LIN {X -0.050,Y -603.917,Z 1305.029,A 0.000,B 0.000,C 90.000,E1 41.148} C_DIS
LIN {X -0.165,Y -603.300,Z 1305.021,A 0.000,B 0.000,C 90.000,E1 39.850} C_DIS
LIN {X 0.003,Y -602.782,Z 1305.016,A 0.000,B 0.000,C 90.000,E1 38.785} C_DIS
LIN {X 0.042,Y -602.471,Z 1305.013,A 0.000,B 0.000,C 90.000,E1 38.257} C_DIS
LIN {X -0.014,Y -601.272,Z 1305.005,A 0.000,B 0.000,C 90.000,E1 36.950} C_DIS
LIN {X 0.141,Y -599.989,Z 1305.000,A 0.000,B 0.000,C 90.000,E1 35.884} C_DIS
LIN {X 0.275,Y -598.512,Z 1304.994,A 0.000,B 0.000,C 90.000,E1 34.818} C_DIS
LIN {X 0.273,Y -596.215,Z 1304.986,A 0.000,B 0.000,C 90.000,E1 33.499} C_DIS
LIN {X -0.207,Y -594.487,Z 1304.982,A 0.000,B 0.000,C 90.000,E1 32.752} C_DIS
LIN {X 0.007,Y -591.783,Z 1304.976,A 0.000,B 0.000,C 90.000,E1 31.671} C_DIS
LIN {X -0.010,Y -589.415,Z 1304.972,A 0.000,B 0.000,C 90.000,E1 30.875} C_DIS
LIN {X -0.049,Y -586.731,Z 1304.967,A 0.000,B 0.000,C 90.000,E1 30.079} C_DIS
LIN {X -0.115,Y -583.665,Z 1304.963,A 0.000,B 0.000,C 90.000,E1 29.283} C_DIS
LIN {X -0.216,Y -580.058,Z 1304.958,A 0.000,B 0.000,C 90.000,E1 28.487} C_DIS
LIN {X 0.289,Y -577.403,Z 1304.955,A 0.000,B 0.000,C 90.000,E1 27.897} C_DIS
LIN {X -0.238,Y -572.396,Z 1304.950,A 0.000,B 0.000,C 90.000,E1 27.001} C_DIS
LIN {X -0.051,Y -569.282,Z 1304.947,A 0.000,B 0.000,C 90.000,E1 26.437} C_DIS
LIN {X 0.274,Y -564.919,Z 1304.943,A 0.000,B 0.000,C 90.000,E1 25.720} C_DIS
LIN {X -0.101,Y -561.279,Z 1304.940,A 0.000,B 0.000,C 90.000,E1 25.207} C_DIS
LIN {X 0.009,Y -557.381,Z 1304.937,A 0.000,B 0.000,C 90.000,E1 24.643} C_DIS
LIN {X 0.090,Y -553.159,Z 1304.934,A 0.000,B 0.000,C 90.000,E1 24.079} C_DIS
LIN {X -0.098,Y -546.387,Z 1304.929,A 0.000,B 0.000,C 90.000,E1 23.259} C_DIS
LIN {X 0.140,Y -539.069,Z 1304.925,A 0.000,B 0.000,C 90.000,E1 22.386} C_DIS
LIN {X 0.134,Y -531.413,Z 1304.920,A 0.000,B 0.000,C 90.000,E1 21.535} C_DIS
LIN {X 0.190,Y -522.299,Z 1304.914,A 0.000,B 0.000,C 90.000,E1 20.556} C_DIS
LIN {X -0.102,Y -511.906,Z 1304.908,A 0.000,B 0.000,C 90.000,E1 19.504} C_DIS
LIN {X -0.036,Y -501.097,Z 1304.902,A 0.000,B 0.000,C 90.000,E1 18.417} C_DIS
LIN {X 0.246,Y -491.595,Z 1304.897,A 0.000,B 0.000,C 90.000,E1 17.457} C_DIS
LIN {X 0.090,Y -484.623,Z 1304.893,A 0.000,B 0.000,C 90.000,E1 16.804} C_DIS
LIN {X -0.137,Y -474.406,Z 1304.888,A 0.000,B 0.000,C 90.000,E1 15.898} C_DIS
LIN {X -0.208,Y -456.704,Z 1304.879,A 0.000,B 0.000,C 90.000,E1 14.300} C_DIS
LIN {X -0.186,Y -437.759,Z 1304.869,A 0.000,B 0.000,C 90.000,E1 12.479} C_DIS
LIN {X -0.013,Y -422.193,Z 1304.860,A 0.000,B 0.000,C 90.000,E1 10.838} C_DIS
LIN {X 0.090,Y -407.857,Z 1304.852,A 0.000,B 0.000,C 90.000,E1 9.265} C_DIS
LIN {X 0.033,Y -398.123,Z 1304.845,A 0.000,B 0.000,C 90.000,E1 8.163} C_DIS
LIN {X 0.181,Y -395.332,Z 1304.843,A 0.000,B 0.000,C 90.000,E1 7.701} C_DIS
LIN {X 0.144,Y -395.311,Z 1304.843,A 0.000,B 0.000,C 90.000,E1 7.701} C_DIS
LIN {X 0.016,Y -396.035,Z 1304.842,A 0.000,B 0.000,C 90.000,E1 7.587} C_DIS
LIN {X 0.131,Y -399.018,Z 1304.841,A 0.000,B 0.000,C 90.000,E1 7.296} C_DIS
LIN {X 0.105,Y -403.349,Z 1304.839,A 0.000,B 0.000,C 90.000,E1 7.004} C_DIS
LIN {X 0.156,Y -411.713,Z 1304.836,A 0.000,B 0.000,C 90.000,E1 6.486} C_DIS
LIN {X -0.092,Y -416.700,Z 1304.834,A 0.000,B 0.000,C 90.000,E1 6.201} C_DIS
LIN {X 0.017,Y -424.463,Z 1304.831,A 0.000,B 0.000,C 90.000,E1 5.625} C_DIS
LIN {X 0.127,Y -430.373,Z 1304.829,A 0.000,B 0.000,C 90.000,E1 5.163} C_DIS
LIN {X -0.129,Y -436.534,Z 1304.826,A 0.000,B 0.000,C 90.000,E1 4.702} C_DIS
LIN {X -0.025,Y -442.431,Z 1304.823,A 0.000,B 0.000,C 90.000,E1 4.188} C_DIS
LIN {X -0.020,Y -451.215,Z 1304.819,A 0.000,B 0.000,C 90.000,E1 3.383} C_DIS
LIN {X -0.087,Y -458.495,Z 1304.815,A 0.000,B 0.000,C 90.000,E1 2.694} C_DIS
LIN {X 0.177,Y -462.637,Z 1304.813,A 0.000,B 0.000,C 90.000,E1 2.236} C_DIS
LIN {X -0.159,Y -466.774,Z 1304.810,A 0.000,B 0.000,C 90.000,E1 1.835} C_DIS
LIN {X 0.206,Y -473.385,Z 1304.806,A 0.000,B 0.000,C 90.000,E1 1.031} C_DIS
LIN {X 0.238,Y -480.443,Z 1304.801,A 0.000,B 0.000,C 90.000,E1 0.115} C_DIS
LIN {X 0.149,Y -486.189,Z 1304.796,A 0.000,B 0.000,C 90.000,E1 359.312} C_DIS
LIN {X -0.196,Y -490.310,Z 1304.793,A 0.000,B 0.000,C 90.000,E1 358.740} C_DIS
LIN {X -0.156,Y -495.830,Z 1304.788,A 0.000,B 0.000,C 90.000,E1 357.822} C_DIS
LIN {X -0.258,Y -500.125,Z 1304.784,A 0.000,B 0.000,C 90.000,E1 357.078} C_DIS
LIN {X 0.016,Y -503.396,Z 1304.780,A 0.000,B 0.000,C 90.000,E1 356.445} C_DIS
LIN {X 0.212,Y -507.901,Z 1304.775,A 0.000,B 0.000,C 90.000,E1 355.527} C_DIS
LIN {X 0.046,Y -510.758,Z 1304.772,A 0.000,B 0.000,C 90.000,E1 354.951} C_DIS
LIN {X 0.075,Y -515.367,Z 1304.766,A 0.000,B 0.000,C 90.000,E1 353.913} C_DIS
LIN {X 0.179,Y -518.468,Z 1304.762,A 0.000,B 0.000,C 90.000,E1 353.166} C_DIS
LIN {X 0.075,Y -521.724,Z 1304.757,A 0.000,B 0.000,C 90.000,E1 352.299} C_DIS
LIN {X 0.004,Y -524.770,Z 1304.752,A 0.000,B 0.000,C 90.000,E1 351.432} C_DIS
LIN {X 0.029,Y -526.616,Z 1304.749,A 0.000,B 0.000,C 90.000,E1 350.849} C_DIS
LIN {X 0.037,Y -530.025,Z 1304.743,A 0.000,B 0.000,C 90.000,E1 349.690} C_DIS
LIN {X 0.186,Y -533.032,Z 1304.736,A 0.000,B 0.000,C 90.000,E1 348.522} C_DIS
LIN {X -0.145,Y -535.534,Z 1304.730,A 0.000,B 0.000,C 90.000,E1 347.409} C_DIS
LIN {X 0.203,Y -537.708,Z 1304.724,A 0.000,B 0.000,C 90.000,E1 346.228} C_DIS
LIN {X -0.198,Y -538.656,Z 1304.720,A 0.000,B 0.000,C 90.000,E1 345.700} C_DIS
LIN {X 0.129,Y -539.857,Z 1304.716,A 0.000,B 0.000,C 90.000,E1 344.810} C_DIS
LIN {X -0.051,Y -540.812,Z 1304.711,A 0.000,B 0.000,C 90.000,E1 343.976} C_DIS
LIN {X -0.221,Y -541.514,Z 1304.706,A 0.000,B 0.000,C 90.000,E1 343.142} C_DIS
LIN {X -0.160,Y -542.045,Z 1304.700,A 0.000,B 0.000,C 90.000,E1 342.000} C_DIS
LIN {X -0.152,Y -542.178,Z 1304.695,A 0.000,B 0.000,C 90.000,E1 341.148} C_DIS
LIN {X 0.143,Y -541.576,Z 1304.687,A 0.000,B 0.000,C 90.000,E1 339.699} C_DIS
LIN {X 0.104,Y -541.174,Z 1304.684,A 0.000,B 0.000,C 90.000,E1 339.135} C_DIS
LIN {X 0.100,Y -540.128,Z 1304.679,A 0.000,B 0.000,C 90.000,E1 338.284} C_DIS
LIN {X 0.285,Y -539.018,Z 1304.675,A 0.000,B 0.000,C 90.000,E1 337.411} C_DIS
LIN {X -0.249,Y -537.510,Z 1304.670,A 0.000,B 0.000,C 90.000,E1 336.613} C_DIS
LIN {X -0.095,Y -535.614,Z 1304.665,A 0.000,B 0.000,C 90.000,E1 335.741} C_DIS
LIN {X 0.113,Y -534.713,Z 1304.664,A 0.000,B 0.000,C 90.000,E1 335.433} C_DIS
LIN {X 0.258,Y -533.249,Z 1304.660,A 0.000,B 0.000,C 90.000,E1 334.845} C_DIS
LIN {X -0.121,Y -530.563,Z 1304.656,A 0.000,B 0.000,C 90.000,E1 334.024} C_DIS
LIN {X 0.043,Y -525.851,Z 1304.648,A 0.000,B 0.000,C 90.000,E1 332.564} C_DIS
LIN {X 0.069,Y -522.798,Z 1304.643,A 0.000,B 0.000,C 90.000,E1 331.691} C_DIS
LIN {X -0.051,Y -518.431,Z 1304.636,A 0.000,B 0.000,C 90.000,E1 330.539} C_DIS
LIN {X -0.013,Y -516.123,Z 1304.633,A 0.000,B 0.000,C 90.000,E1 329.950} C_DIS
LIN {X -0.084,Y -512.267,Z 1304.628,A 0.000,B 0.000,C 90.000,E1 329.076} C_DIS
LIN {X -0.112,Y -507.612,Z 1304.622,A 0.000,B 0.000,C 90.000,E1 328.043} C_DIS
LIN {X -0.156,Y -501.579,Z 1304.615,A 0.000,B 0.000,C 90.000,E1 326.707} C_DIS
LIN {X 0.020,Y -499.293,Z 1304.612,A 0.000,B 0.000,C 90.000,E1 326.087} C_DIS
LIN {X -0.104,Y -498.271,Z 1304.610,A 0.000,B 0.000,C 90.000,E1 325.801} C_DIS
LIN {X -0.085,Y -496.074,Z 1304.605,A 0.000,B 0.000,C 90.000,E1 324.895} C_DIS
LIN {X -0.093,Y -494.546,Z 1304.600,A 0.000,B 0.000,C 90.000,E1 323.989} C_DIS
LIN {X 0.029,Y -493.279,Z 1304.593,A 0.000,B 0.000,C 90.000,E1 322.763} C_DIS
LIN {X -0.017,Y -492.454,Z 1304.585,A 0.000,B 0.000,C 90.000,E1 321.251} C_DIS
LIN {X -0.303,Y -492.309,Z 1304.575,A 0.000,B 0.000,C 90.000,E1 319.461} C_DIS
LIN {X -0.124,Y -491.974,Z 1304.570,A 0.000,B 0.000,C 90.000,E1 318.528} C_DIS
LIN {X -0.113,Y -491.483,Z 1304.566,A 0.000,B 0.000,C 90.000,E1 317.919} C_DIS
LIN {X -0.108,Y -490.622,Z 1304.563,A 0.000,B 0.000,C 90.000,E1 317.310} C_DIS
LIN {X 0.059,Y -489.988,Z 1304.561,A 0.000,B 0.000,C 90.000,E1 316.986} C_DIS
LIN {X -0.111,Y -489.131,Z 1304.559,A 0.000,B 0.000,C 90.000,E1 316.701} C_DIS
LIN {X -0.030,Y -488.569,Z 1304.559,A 0.000,B 0.000,C 90.000,E1 316.539} C_DIS
LIN {X 0.051,Y -487.839,Z 1304.558,A 0.000,B 0.000,C 90.000,E1 316.377} C_DIS
LIN {X 0.129,Y -486.724,Z 1304.557,A 0.000,B 0.000,C 90.000,E1 316.215} C_DIS
LIN {X -0.012,Y -466.023,Z 1304.543,A 0.000,B 0.000,C 90.000,E1 313.785} C_DIS
LIN {X -0.005,Y -447.038,Z 1304.529,A 0.000,B 0.000,C 90.000,E1 311.229} C_DIS
LIN {X 0.097,Y -429.911,Z 1304.515,A 0.000,B 0.000,C 90.000,E1 308.588} C_DIS
LIN {X 0.152,Y -414.520,Z 1304.500,A 0.000,B 0.000,C 90.000,E1 305.884} C_DIS
LIN {X -0.152,Y -400.749,Z 1304.484,A 0.000,B 0.000,C 90.000,E1 303.166} C_DIS
LIN {X 0.025,Y -393.605,Z 1304.475,A 0.000,B 0.000,C 90.000,E1 301.544} C_DIS
LIN {X -0.013,Y -393.590,Z 1304.475,A 0.000,B 0.000,C 90.000,E1 301.544} C_DIS
LIN {X -0.052,Y -396.754,Z 1304.460,A 0.000,B 0.000,C 90.000,E1 298.743} C_DIS
LIN {X 0.167,Y -397.096,Z 1304.458,A 0.000,B 0.000,C 90.000,E1 298.359} C_DIS
LIN {X -0.047,Y -401.546,Z 1304.427,A 0.000,B 0.000,C 90.000,E1 292.770} C_DIS
LIN {X 0.016,Y -404.021,Z 1304.399,A 0.000,B 0.000,C 90.000,E1 287.873} C_DIS
LIN {X 0.094,Y -404.611,Z 1304.396,A 0.000,B 0.000,C 90.000,E1 287.166} C_DIS
LIN {X -0.191,Y -404.756,Z 1304.394,A 0.000,B 0.000,C 90.000,E1 286.858} C_DIS
LIN {X 0.195,Y -406.069,Z 1304.365,A 0.000,B 0.000,C 90.000,E1 281.591} C_DIS
LIN {X 0.203,Y -406.117,Z 1304.363,A 0.000,B 0.000,C 90.000,E1 281.243} C_DIS
LIN {X -0.164,Y -405.668,Z 1304.334,A 0.000,B 0.000,C 90.000,E1 276.087} C_DIS
LIN {X -0.160,Y -405.564,Z 1304.332,A 0.000,B 0.000,C 90.000,E1 275.739} C_DIS
LIN {X -0.085,Y -403.529,Z 1304.305,A 0.000,B 0.000,C 90.000,E1 270.859} C_DIS
LIN {X -0.118,Y -403.319,Z 1304.303,A 0.000,B 0.000,C 90.000,E1 270.516} C_DIS
LIN {X 0.070,Y -398.979,Z 1304.272,A 0.000,B 0.000,C 90.000,E1 264.894} C_DIS
LIN {X -0.124,Y -393.151,Z 1304.242,A 0.000,B 0.000,C 90.000,E1 259.634} C_DIS
LIN {X -0.091,Y -392.885,Z 1304.240,A 0.000,B 0.000,C 90.000,E1 259.275} C_DIS
LIN {X 0.064,Y -388.626,Z 1304.225,A 0.000,B 0.000,C 90.000,E1 256.408} C_DIS
LIN {X -0.023,Y -385.321,Z 1304.209,A 0.000,B 0.000,C 90.000,E1 253.559} C_DIS
LIN {X -0.002,Y -384.870,Z 1304.207,A 0.000,B 0.000,C 90.000,E1 253.196} C_DIS
LIN {X 0.101,Y -378.044,Z 1304.183,A 0.000,B 0.000,C 90.000,E1 248.847} C_DIS
LIN {X -0.023,Y -376.296,Z 1304.175,A 0.000,B 0.000,C 90.000,E1 247.411} C_DIS
LIN {X -0.043,Y -375.749,Z 1304.172,A 0.000,B 0.000,C 90.000,E1 247.050} C_DIS
LIN {X -0.038,Y -371.592,Z 1304.160,A 0.000,B 0.000,C 90.000,E1 244.717} C_DIS
LIN {X -0.075,Y -371.601,Z 1304.160,A 0.000,B 0.000,C 90.000,E1 244.717} C_DIS
LIN {X -0.178,Y -381.741,Z 1304.143,A 0.000,B 0.000,C 90.000,E1 241.769} C_DIS
LIN {X 0.018,Y -393.143,Z 1304.127,A 0.000,B 0.000,C 90.000,E1 238.869} C_DIS
LIN {X -0.206,Y -406.022,Z 1304.111,A 0.000,B 0.000,C 90.000,E1 236.087} C_DIS
LIN {X 0.118,Y -420.472,Z 1304.096,A 0.000,B 0.000,C 90.000,E1 233.290} C_DIS
LIN {X -0.129,Y -435.544,Z 1304.082,A 0.000,B 0.000,C 90.000,E1 230.803} C_DIS
LIN {X 0.009,Y -447.590,Z 1304.072,A 0.000,B 0.000,C 90.000,E1 228.976} C_DIS
LIN {X 0.043,Y -448.501,Z 1304.071,A 0.000,B 0.000,C 90.000,E1 228.809} C_DIS
LIN {X 0.031,Y -449.596,Z 1304.069,A 0.000,B 0.000,C 90.000,E1 228.485} C_DIS
LIN {X 0.025,Y -450.299,Z 1304.068,A 0.000,B 0.000,C 90.000,E1 228.162} C_DIS
LIN {X 0.028,Y -451.192,Z 1304.064,A 0.000,B 0.000,C 90.000,E1 227.514} C_DIS
LIN {X 0.065,Y -451.741,Z 1304.060,A 0.000,B 0.000,C 90.000,E1 226.863} C_DIS
LIN {X 0.083,Y -452.049,Z 1304.057,A 0.000,B 0.000,C 90.000,E1 226.215} C_DIS
LIN {X 0.118,Y -452.180,Z 1304.052,A 0.000,B 0.000,C 90.000,E1 225.243} C_DIS
LIN {X -0.096,Y -452.123,Z 1304.037,A 0.000,B 0.000,C 90.000,E1 222.690} C_DIS
LIN {X 0.191,Y -453.631,Z 1304.014,A 0.000,B 0.000,C 90.000,E1 218.463} C_DIS
LIN {X -0.015,Y -454.594,Z 1304.007,A 0.000,B 0.000,C 90.000,E1 217.202} C_DIS
LIN {X 0.058,Y -456.363,Z 1303.994,A 0.000,B 0.000,C 90.000,E1 214.945} C_DIS
LIN {X 0.018,Y -459.450,Z 1303.976,A 0.000,B 0.000,C 90.000,E1 211.750} C_DIS
LIN {X 0.125,Y -462.952,Z 1303.961,A 0.000,B 0.000,C 90.000,E1 208.871} C_DIS
LIN {X 0.072,Y -466.804,Z 1303.945,A 0.000,B 0.000,C 90.000,E1 206.027} C_DIS
LIN {X 0.115,Y -469.582,Z 1303.934,A 0.000,B 0.000,C 90.000,E1 204.131} C_DIS
LIN {X -0.113,Y -471.829,Z 1303.925,A 0.000,B 0.000,C 90.000,E1 202.589} C_DIS
LIN {X 0.093,Y -474.922,Z 1303.913,A 0.000,B 0.000,C 90.000,E1 200.375} C_DIS
LIN {X -0.214,Y -477.865,Z 1303.903,A 0.000,B 0.000,C 90.000,E1 198.544} C_DIS
LIN {X -0.165,Y -480.689,Z 1303.893,A 0.000,B 0.000,C 90.000,E1 196.677} C_DIS
LIN {X -0.194,Y -483.514,Z 1303.882,A 0.000,B 0.000,C 90.000,E1 194.828} C_DIS
LIN {X 0.182,Y -486.378,Z 1303.872,A 0.000,B 0.000,C 90.000,E1 192.939} C_DIS
LIN {X -0.176,Y -489.564,Z 1303.860,A 0.000,B 0.000,C 90.000,E1 190.838} C_DIS
LIN {X 0.135,Y -492.263,Z 1303.850,A 0.000,B 0.000,C 90.000,E1 188.973} C_DIS
LIN {X 0.032,Y -494.499,Z 1303.842,A 0.000,B 0.000,C 90.000,E1 187.466} C_DIS
LIN {X -0.246,Y -497.138,Z 1303.831,A 0.000,B 0.000,C 90.000,E1 185.682} C_DIS
LIN {X 0.131,Y -499.224,Z 1303.823,A 0.000,B 0.000,C 90.000,E1 184.131} C_DIS
LIN {X -0.077,Y -501.405,Z 1303.813,A 0.000,B 0.000,C 90.000,E1 182.350} C_DIS
LIN {X 0.081,Y -502.384,Z 1303.808,A 0.000,B 0.000,C 90.000,E1 181.432} C_DIS
LIN {X 0.013,Y -503.892,Z 1303.800,A 0.000,B 0.000,C 90.000,E1 179.943} C_DIS
LIN {X -0.030,Y -505.128,Z 1303.791,A 0.000,B 0.000,C 90.000,E1 178.453} C_DIS
LIN {X 0.064,Y -505.791,Z 1303.785,A 0.000,B 0.000,C 90.000,E1 177.249} C_DIS
LIN {X -0.228,Y -506.243,Z 1303.780,A 0.000,B 0.000,C 90.000,E1 176.388} C_DIS
LIN {X -0.011,Y -506.464,Z 1303.775,A 0.000,B 0.000,C 90.000,E1 175.469} C_DIS
LIN {X 0.141,Y -506.569,Z 1303.768,A 0.000,B 0.000,C 90.000,E1 174.261} C_DIS
LIN {X 0.233,Y -506.299,Z 1303.760,A 0.000,B 0.000,C 90.000,E1 172.761} C_DIS
LIN {X 0.177,Y -506.226,Z 1303.758,A 0.000,B 0.000,C 90.000,E1 172.470} C_DIS
LIN {X -0.112,Y -505.418,Z 1303.752,A 0.000,B 0.000,C 90.000,E1 171.310} C_DIS
LIN {X 0.140,Y -504.482,Z 1303.747,A 0.000,B 0.000,C 90.000,E1 170.387} C_DIS
LIN {X -0.033,Y -503.442,Z 1303.742,A 0.000,B 0.000,C 90.000,E1 169.511} C_DIS
LIN {X -0.214,Y -502.103,Z 1303.737,A 0.000,B 0.000,C 90.000,E1 168.634} C_DIS
LIN {X -0.063,Y -499.175,Z 1303.728,A 0.000,B 0.000,C 90.000,E1 167.117} C_DIS
LIN {X -0.182,Y -497.026,Z 1303.723,A 0.000,B 0.000,C 90.000,E1 166.228} C_DIS
LIN {X 0.161,Y -494.687,Z 1303.718,A 0.000,B 0.000,C 90.000,E1 165.283} C_DIS
LIN {X -0.109,Y -491.352,Z 1303.712,A 0.000,B 0.000,C 90.000,E1 164.102} C_DIS
LIN {X 0.170,Y -487.684,Z 1303.705,A 0.000,B 0.000,C 90.000,E1 162.851} C_DIS
LIN {X 0.064,Y -484.249,Z 1303.700,A 0.000,B 0.000,C 90.000,E1 161.945} C_DIS
LIN {X 0.071,Y -482.858,Z 1303.698,A 0.000,B 0.000,C 90.000,E1 161.638} C_DIS
LIN {X -0.083,Y -479.965,Z 1303.695,A 0.000,B 0.000,C 90.000,E1 161.040} C_DIS
LIN {X -0.117,Y -476.057,Z 1303.689,A 0.000,B 0.000,C 90.000,E1 160.115} C_DIS
LIN {X 0.121,Y -473.758,Z 1303.686,A 0.000,B 0.000,C 90.000,E1 159.464} C_DIS
LIN {X 0.093,Y -472.774,Z 1303.684,A 0.000,B 0.000,C 90.000,E1 159.156} C_DIS
LIN {X 0.060,Y -472.032,Z 1303.683,A 0.000,B 0.000,C 90.000,E1 158.847} C_DIS
LIN {X 0.025,Y -471.480,Z 1303.681,A 0.000,B 0.000,C 90.000,E1 158.539} C_DIS
LIN {X -0.251,Y -471.076,Z 1303.678,A 0.000,B 0.000,C 90.000,E1 158.103} C_DIS
LIN {X -0.139,Y -471.938,Z 1303.675,A 0.000,B 0.000,C 90.000,E1 157.486} C_DIS
LIN {X 0.193,Y -473.245,Z 1303.674,A 0.000,B 0.000,C 90.000,E1 157.230} C_DIS
LIN {X -0.004,Y -474.581,Z 1303.672,A 0.000,B 0.000,C 90.000,E1 156.922} C_DIS
LIN {X -0.076,Y -475.911,Z 1303.671,A 0.000,B 0.000,C 90.000,E1 156.794} C_DIS
LIN {X 0.093,Y -478.294,Z 1303.669,A 0.000,B 0.000,C 90.000,E1 156.485} C_DIS
LIN {X -0.107,Y -488.174,Z 1303.665,A 0.000,B 0.000,C 90.000,E1 155.665} C_DIS
LIN {X -0.025,Y -495.221,Z 1303.661,A 0.000,B 0.000,C 90.000,E1 155.025} C_DIS
LIN {X 0.094,Y -500.828,Z 1303.658,A 0.000,B 0.000,C 90.000,E1 154.485} C_DIS
LIN {X 0.076,Y -504.805,Z 1303.656,A 0.000,B 0.000,C 90.000,E1 154.101} C_DIS
LIN {X 0.211,Y -511.243,Z 1303.652,A 0.000,B 0.000,C 90.000,E1 153.384} C_DIS
LIN {X -0.244,Y -515.035,Z 1303.650,A 0.000,B 0.000,C 90.000,E1 152.999} C_DIS
LIN {X 0.224,Y -519.713,Z 1303.647,A 0.000,B 0.000,C 90.000,E1 152.359} C_DIS
LIN {X 0.271,Y -523.864,Z 1303.643,A 0.000,B 0.000,C 90.000,E1 151.769} C_DIS
LIN {X -0.111,Y -527.497,Z 1303.640,A 0.000,B 0.000,C 90.000,E1 151.229} C_DIS
LIN {X -0.264,Y -530.566,Z 1303.637,A 0.000,B 0.000,C 90.000,E1 150.667} C_DIS
LIN {X -0.140,Y -533.050,Z 1303.634,A 0.000,B 0.000,C 90.000,E1 150.078} C_DIS
LIN {X 0.001,Y -535.130,Z 1303.630,A 0.000,B 0.000,C 90.000,E1 149.488} C_DIS
LIN {X -0.018,Y -536.121,Z 1303.629,A 0.000,B 0.000,C 90.000,E1 149.203} C_DIS
LIN {X 0.144,Y -537.716,Z 1303.626,A 0.000,B 0.000,C 90.000,E1 148.614} C_DIS
LIN {X -0.139,Y -539.753,Z 1303.621,A 0.000,B 0.000,C 90.000,E1 147.788} C_DIS
LIN {X 0.044,Y -540.924,Z 1303.618,A 0.000,B 0.000,C 90.000,E1 147.199} C_DIS
LIN {X -0.083,Y -541.922,Z 1303.615,A 0.000,B 0.000,C 90.000,E1 146.786} C_DIS
LIN {X -0.340,Y -542.024,Z 1303.615,A 0.000,B 0.000,C 90.000,E1 146.707} C_DIS
LIN {X 0.364,Y -543.123,Z 1303.614,A 0.000,B 0.000,C 90.000,E1 146.421} C_DIS
LIN {X 0.182,Y -543.846,Z 1303.612,A 0.000,B 0.000,C 90.000,E1 146.215} C_DIS
LIN {X 0.254,Y -546.623,Z 1303.611,A 0.000,B 0.000,C 90.000,E1 146.008} C_DIS
LIN {X -0.044,Y -547.860,Z 1303.611,A 0.000,B 0.000,C 90.000,E1 145.928} C_DIS
LIN {X 0.074,Y -553.909,Z 1303.609,A 0.000,B 0.000,C 90.000,E1 145.595} C_DIS
LIN {X -0.289,Y -559.106,Z 1303.608,A 0.000,B 0.000,C 90.000,E1 145.388} C_DIS
LIN {X 0.100,Y -565.147,Z 1303.606,A 0.000,B 0.000,C 90.000,E1 145.022} C_DIS
LIN {X 0.080,Y -572.943,Z 1303.603,A 0.000,B 0.000,C 90.000,E1 144.562} C_DIS
LIN {X 0.054,Y -577.273,Z 1303.602,A 0.000,B 0.000,C 90.000,E1 144.276} C_DIS
LIN {X 0.184,Y -585.796,Z 1303.598,A 0.000,B 0.000,C 90.000,E1 143.623} C_DIS
LIN {X 0.036,Y -588.557,Z 1303.597,A 0.000,B 0.000,C 90.000,E1 143.417} C_DIS
LIN {X 0.216,Y -593.907,Z 1303.594,A 0.000,B 0.000,C 90.000,E1 142.924} C_DIS
LIN {X 0.178,Y -597.765,Z 1303.592,A 0.000,B 0.000,C 90.000,E1 142.557} C_DIS
LIN {X 0.020,Y -601.414,Z 1303.590,A 0.000,B 0.000,C 90.000,E1 142.190} C_DIS
LIN {X 0.075,Y -605.960,Z 1303.587,A 0.000,B 0.000,C 90.000,E1 141.662} C_DIS
LIN {X 0.285,Y -609.166,Z 1303.585,A 0.000,B 0.000,C 90.000,E1 141.251} C_DIS
LIN {X -0.208,Y -614.828,Z 1303.581,A 0.000,B 0.000,C 90.000,E1 140.517} C_DIS
LIN {X -0.087,Y -618.352,Z 1303.578,A 0.000,B 0.000,C 90.000,E1 139.989} C_DIS
LIN {X -0.093,Y -623.243,Z 1303.573,A 0.000,B 0.000,C 90.000,E1 139.218} C_DIS
LIN {X 0.049,Y -627.022,Z 1303.570,A 0.000,B 0.000,C 90.000,E1 138.566} C_DIS
LIN {X 0.170,Y -630.521,Z 1303.566,A 0.000,B 0.000,C 90.000,E1 137.919} C_DIS
LIN {X -0.210,Y -635.065,Z 1303.561,A 0.000,B 0.000,C 90.000,E1 137.067} C_DIS
LIN {X -0.139,Y -639.970,Z 1303.556,A 0.000,B 0.000,C 90.000,E1 136.053} C_DIS
LIN {X -0.015,Y -644.817,Z 1303.550,A 0.000,B 0.000,C 90.000,E1 135.040} C_DIS
LIN {X 0.115,Y -650.599,Z 1303.543,A 0.000,B 0.000,C 90.000,E1 133.785} C_DIS
LIN {X -0.088,Y -655.199,Z 1303.538,A 0.000,B 0.000,C 90.000,E1 132.813} C_DIS
LIN {X -0.227,Y -660.734,Z 1303.531,A 0.000,B 0.000,C 90.000,E1 131.595} C_DIS
LIN {X 0.196,Y -663.953,Z 1303.527,A 0.000,B 0.000,C 90.000,E1 130.825} C_DIS
LIN {X 0.220,Y -667.031,Z 1303.523,A 0.000,B 0.000,C 90.000,E1 130.092} C_DIS
LIN {X 0.274,Y -670.906,Z 1303.517,A 0.000,B 0.000,C 90.000,E1 129.116} C_DIS
LIN {X -0.043,Y -675.316,Z 1303.511,A 0.000,B 0.000,C 90.000,E1 127.935} C_DIS
LIN {X 0.087,Y -677.032,Z 1303.508,A 0.000,B 0.000,C 90.000,E1 127.443} C_DIS
LIN {X -0.157,Y -680.026,Z 1303.503,A 0.000,B 0.000,C 90.000,E1 126.503} C_DIS
LIN {X 0.185,Y -682.841,Z 1303.497,A 0.000,B 0.000,C 90.000,E1 125.518} C_DIS
LIN {X 0.187,Y -685.958,Z 1303.491,A 0.000,B 0.000,C 90.000,E1 124.326} C_DIS
LIN {X 0.019,Y -687.660,Z 1303.487,A 0.000,B 0.000,C 90.000,E1 123.627} C_DIS
LIN {X 0.064,Y -689.175,Z 1303.483,A 0.000,B 0.000,C 90.000,E1 122.911} C_DIS
LIN {X 0.377,Y -691.672,Z 1303.475,A 0.000,B 0.000,C 90.000,E1 121.465} C_DIS
LIN {X -0.234,Y -693.463,Z 1303.469,A 0.000,B 0.000,C 90.000,E1 120.335} C_DIS
LIN {X 0.143,Y -694.767,Z 1303.463,A 0.000,B 0.000,C 90.000,E1 119.361} C_DIS
LIN {X -0.065,Y -695.790,Z 1303.458,A 0.000,B 0.000,C 90.000,E1 118.437} C_DIS
LIN {X 0.090,Y -696.330,Z 1303.454,A 0.000,B 0.000,C 90.000,E1 117.719} C_DIS
LIN {X 0.247,Y -696.649,Z 1303.450,A 0.000,B 0.000,C 90.000,E1 117.001} C_DIS
LIN {X -0.272,Y -696.762,Z 1303.445,A 0.000,B 0.000,C 90.000,E1 116.104} C_DIS
LIN {X -0.124,Y -696.410,Z 1303.441,A 0.000,B 0.000,C 90.000,E1 115.387} C_DIS
LIN {X 0.094,Y -696.014,Z 1303.438,A 0.000,B 0.000,C 90.000,E1 114.899} C_DIS
LIN {X -0.317,Y -695.198,Z 1303.436,A 0.000,B 0.000,C 90.000,E1 114.463} C_DIS
LIN {X -0.063,Y -694.612,Z 1303.434,A 0.000,B 0.000,C 90.000,E1 114.207} C_DIS
LIN {X 0.157,Y -693.038,Z 1303.432,A 0.000,B 0.000,C 90.000,E1 113.718} C_DIS
LIN {X -0.112,Y -690.937,Z 1303.430,A 0.000,B 0.000,C 90.000,E1 113.387} C_DIS
LIN {X 0.123,Y -689.475,Z 1303.429,A 0.000,B 0.000,C 90.000,E1 113.131} C_DIS
LIN {X -0.032,Y -688.451,Z 1303.428,A 0.000,B 0.000,C 90.000,E1 113.025} C_DIS
LIN {X 0.083,Y -686.952,Z 1303.427,A 0.000,B 0.000,C 90.000,E1 112.898} C_DIS
LIN {X 0.028,Y -682.434,Z 1303.426,A 0.000,B 0.000,C 90.000,E1 112.589} C_DIS
LIN {X -0.301,Y -679.515,Z 1303.425,A 0.000,B 0.000,C 90.000,E1 112.461} C_DIS
LIN {X 0.110,Y -672.799,Z 1303.423,A 0.000,B 0.000,C 90.000,E1 112.206} C_DIS
LIN {X 0.177,Y -665.491,Z 1303.423,A 0.000,B 0.000,C 90.000,E1 112.078} C_DIS
LIN {X -0.131,Y -663.364,Z 1303.423,A 0.000,B 0.000,C 90.000,E1 112.078} C_DIS
LIN {X -0.109,Y -653.556,Z 1303.422,A 0.000,B 0.000,C 90.000,E1 112.025} C_DIS
LIN {X -0.245,Y -649.342,Z 1303.422,A 0.000,B 0.000,C 90.000,E1 112.025} C_DIS
LIN {X 0.005,Y -644.465,Z 1303.422,A 0.000,B 0.000,C 90.000,E1 111.950} C_DIS
LIN {X 0.138,Y -642.862,Z 1303.422,A 0.000,B 0.000,C 90.000,E1 111.897} C_DIS
LIN {X 0.123,Y -641.254,Z 1303.422,A 0.000,B 0.000,C 90.000,E1 111.844} C_DIS
LIN {X 0.082,Y -641.206,Z 1303.421,A 0.000,B 0.000,C 90.000,E1 111.844} C_DIS
LIN {X 0.083,Y -642.691,Z 1303.420,A 0.000,B 0.000,C 90.000,E1 111.535} C_DIS
LIN {X -0.265,Y -651.067,Z 1303.414,A 0.000,B 0.000,C 90.000,E1 110.482} C_DIS
LIN {X 0.330,Y -655.258,Z 1303.410,A 0.000,B 0.000,C 90.000,E1 109.812} C_DIS
LIN {X 0.127,Y -658.821,Z 1303.407,A 0.000,B 0.000,C 90.000,E1 109.214} C_DIS
LIN {X 0.169,Y -662.044,Z 1303.403,A 0.000,B 0.000,C 90.000,E1 108.598} C_DIS
LIN {X 0.074,Y -665.312,Z 1303.399,A 0.000,B 0.000,C 90.000,E1 107.873} C_DIS
LIN {X -0.106,Y -667.316,Z 1303.397,A 0.000,B 0.000,C 90.000,E1 107.402} C_DIS
LIN {X -0.151,Y -669.881,Z 1303.393,A 0.000,B 0.000,C 90.000,E1 106.677} C_DIS
LIN {X -0.179,Y -672.033,Z 1303.389,A 0.000,B 0.000,C 90.000,E1 105.953} C_DIS
LIN {X 0.278,Y -673.837,Z 1303.385,A 0.000,B 0.000,C 90.000,E1 105.190} C_DIS
LIN {X 0.111,Y -675.319,Z 1303.380,A 0.000,B 0.000,C 90.000,E1 104.481} C_DIS
LIN {X -0.042,Y -676.585,Z 1303.377,A 0.000,B 0.000,C 90.000,E1 103.772} C_DIS
LIN {X -0.184,Y -677.381,Z 1303.373,A 0.000,B 0.000,C 90.000,E1 103.063} C_DIS
LIN {X -0.321,Y -677.834,Z 1303.369,A 0.000,B 0.000,C 90.000,E1 102.355} C_DIS
LIN {X 0.250,Y -677.943,Z 1303.366,A 0.000,B 0.000,C 90.000,E1 101.827} C_DIS
LIN {X -0.023,Y -677.746,Z 1303.362,A 0.000,B 0.000,C 90.000,E1 101.130} C_DIS
LIN {X -0.119,Y -677.384,Z 1303.359,A 0.000,B 0.000,C 90.000,E1 100.658} C_DIS
LIN {X -0.169,Y -677.169,Z 1303.358,A 0.000,B 0.000,C 90.000,E1 100.423} C_DIS
LIN {X 0.219,Y -676.048,Z 1303.354,A 0.000,B 0.000,C 90.000,E1 99.670} C_DIS
LIN {X -0.007,Y -674.961,Z 1303.351,A 0.000,B 0.000,C 90.000,E1 99.208} C_DIS
LIN {X -0.236,Y -673.584,Z 1303.349,A 0.000,B 0.000,C 90.000,E1 98.746} C_DIS
LIN {X 0.292,Y -671.751,Z 1303.346,A 0.000,B 0.000,C 90.000,E1 98.219} C_DIS
LIN {X 0.044,Y -669.630,Z 1303.343,A 0.000,B 0.000,C 90.000,E1 97.757} C_DIS
LIN {X 0.271,Y -666.001,Z 1303.339,A 0.000,B 0.000,C 90.000,E1 97.011} C_DIS
LIN {X -0.026,Y -662.614,Z 1303.336,A 0.000,B 0.000,C 90.000,E1 96.429} C_DIS
LIN {X -0.306,Y -660.507,Z 1303.334,A 0.000,B 0.000,C 90.000,E1 96.087} C_DIS
LIN {X -0.065,Y -656.443,Z 1303.330,A 0.000,B 0.000,C 90.000,E1 95.454} C_DIS
LIN {X 0.142,Y -651.960,Z 1303.327,A 0.000,B 0.000,C 90.000,E1 94.821} C_DIS
LIN {X -0.229,Y -648.013,Z 1303.324,A 0.000,B 0.000,C 90.000,E1 94.359} C_DIS
LIN {X 0.018,Y -643.717,Z 1303.321,A 0.000,B 0.000,C 90.000,E1 93.841} C_DIS
LIN {X -0.017,Y -636.825,Z 1303.317,A 0.000,B 0.000,C 90.000,E1 93.094} C_DIS
LIN {X 0.005,Y -628.639,Z 1303.313,A 0.000,B 0.000,C 90.000,E1 92.236} C_DIS
LIN {X 0.246,Y -623.618,Z 1303.310,A 0.000,B 0.000,C 90.000,E1 91.718} C_DIS
LIN {X 0.050,Y -615.317,Z 1303.306,A 0.000,B 0.000,C 90.000,E1 91.031} C_DIS
LIN {X -0.244,Y -609.295,Z 1303.303,A 0.000,B 0.000,C 90.000,E1 90.630} C_DIS
LIN {X 0.044,Y -601.368,Z 1303.301,A 0.000,B 0.000,C 90.000,E1 90.115} C_DIS
LIN {X -0.063,Y -594.645,Z 1303.299,A 0.000,B 0.000,C 90.000,E1 89.771} C_DIS
LIN {X -0.158,Y -589.339,Z 1303.297,A 0.000,B 0.000,C 90.000,E1 89.542} C_DIS
LIN {X -0.099,Y -580.328,Z 1303.296,A 0.000,B 0.000,C 90.000,E1 89.198} C_DIS
LIN {X -0.170,Y -576.972,Z 1303.295,A 0.000,B 0.000,C 90.000,E1 89.083} C_DIS
LIN {X -0.257,Y -571.652,Z 1303.294,A 0.000,B 0.000,C 90.000,E1 88.854} C_DIS
LIN {X -0.173,Y -570.221,Z 1303.292,A 0.000,B 0.000,C 90.000,E1 88.625} C_DIS
LIN {X -0.215,Y -570.198,Z 1303.292,A 0.000,B 0.000,C 90.000,E1 88.625} C_DIS
LIN {X -0.068,Y -570.012,Z 1303.290,A 0.000,B 0.000,C 90.000,E1 88.282} C_DIS
LIN {X -0.232,Y -570.505,Z 1303.286,A 0.000,B 0.000,C 90.000,E1 87.478} C_DIS
LIN {X 0.040,Y -571.964,Z 1303.277,A 0.000,B 0.000,C 90.000,E1 85.812} C_DIS
LIN {X 0.088,Y -574.360,Z 1303.265,A 0.000,B 0.000,C 90.000,E1 83.628} C_DIS
LIN {X -0.007,Y -576.220,Z 1303.256,A 0.000,B 0.000,C 90.000,E1 82.008} C_DIS
LIN {X -0.062,Y -578.215,Z 1303.247,A 0.000,B 0.000,C 90.000,E1 80.387} C_DIS
LIN {X 0.139,Y -579.484,Z 1303.241,A 0.000,B 0.000,C 90.000,E1 79.285} C_DIS
LIN {X 0.121,Y -580.839,Z 1303.233,A 0.000,B 0.000,C 90.000,E1 77.937} C_DIS
LIN {X -0.100,Y -581.838,Z 1303.227,A 0.000,B 0.000,C 90.000,E1 76.881} C_DIS
LIN {X 0.062,Y -582.910,Z 1303.220,A 0.000,B 0.000,C 90.000,E1 75.519} C_DIS
LIN {X 0.245,Y -583.849,Z 1303.212,A 0.000,B 0.000,C 90.000,E1 74.157} C_DIS
LIN {X 0.273,Y -584.923,Z 1303.203,A 0.000,B 0.000,C 90.000,E1 72.543} C_DIS
LIN {X -0.055,Y -585.973,Z 1303.194,A 0.000,B 0.000,C 90.000,E1 70.967} C_DIS
LIN {X 0.187,Y -586.974,Z 1303.185,A 0.000,B 0.000,C 90.000,E1 69.337} C_DIS
LIN {X -0.108,Y -587.806,Z 1303.178,A 0.000,B 0.000,C 90.000,E1 68.028} C_DIS
LIN {X 0.051,Y -588.866,Z 1303.169,A 0.000,B 0.000,C 90.000,E1 66.410} C_DIS
LIN {X 0.222,Y -589.936,Z 1303.160,A 0.000,B 0.000,C 90.000,E1 64.793} C_DIS
LIN {X -0.306,Y -590.906,Z 1303.153,A 0.000,B 0.000,C 90.000,E1 63.512} C_DIS
LIN {X -0.218,Y -592.475,Z 1303.142,A 0.000,B 0.000,C 90.000,E1 61.641} C_DIS
LIN {X 0.090,Y -593.782,Z 1303.135,A 0.000,B 0.000,C 90.000,E1 60.284} C_DIS
LIN {X -0.105,Y -595.346,Z 1303.126,A 0.000,B 0.000,C 90.000,E1 58.712} C_DIS
LIN {X 0.163,Y -597.320,Z 1303.116,A 0.000,B 0.000,C 90.000,E1 56.834} C_DIS
LIN {X 0.054,Y -598.990,Z 1303.107,A 0.000,B 0.000,C 90.000,E1 55.261} C_DIS
LIN {X 0.070,Y -600.729,Z 1303.097,A 0.000,B 0.000,C 90.000,E1 53.417} C_DIS
LIN {X 0.240,Y -602.088,Z 1303.088,A 0.000,B 0.000,C 90.000,E1 51.823} C_DIS
LIN {X -0.033,Y -603.238,Z 1303.079,A 0.000,B 0.000,C 90.000,E1 50.275} C_DIS
LIN {X 0.307,Y -604.114,Z 1303.072,A 0.000,B 0.000,C 90.000,E1 48.933} C_DIS
LIN {X -0.048,Y -604.422,Z 1303.066,A 0.000,B 0.000,C 90.000,E1 47.919} C_DIS
LIN {X -0.350,Y -604.685,Z 1303.057,A 0.000,B 0.000,C 90.000,E1 46.377} C_DIS
LIN {X -0.046,Y -604.822,Z 1303.050,A 0.000,B 0.000,C 90.000,E1 45.040} C_DIS
LIN {X -0.399,Y -604.649,Z 1303.044,A 0.000,B 0.000,C 90.000,E1 44.028} C_DIS
LIN {X -0.090,Y -604.311,Z 1303.037,A 0.000,B 0.000,C 90.000,E1 42.690} C_DIS
LIN {X -0.193,Y -603.926,Z 1303.030,A 0.000,B 0.000,C 90.000,E1 41.391} C_DIS
LIN {X -0.303,Y -603.327,Z 1303.023,A 0.000,B 0.000,C 90.000,E1 40.092} C_DIS
LIN {X -0.222,Y -602.845,Z 1303.017,A 0.000,B 0.000,C 90.000,E1 39.036} C_DIS
LIN {X 0.065,Y -602.347,Z 1303.012,A 0.000,B 0.000,C 90.000,E1 38.222} C_DIS
LIN {X -0.004,Y -601.133,Z 1303.005,A 0.000,B 0.000,C 90.000,E1 36.916} C_DIS
LIN {X -0.211,Y -599.847,Z 1302.999,A 0.000,B 0.000,C 90.000,E1 35.884} C_DIS
LIN {X -0.078,Y -598.349,Z 1302.993,A 0.000,B 0.000,C 90.000,E1 34.818} C_DIS
LIN {X -0.309,Y -596.553,Z 1302.988,A 0.000,B 0.000,C 90.000,E1 33.785} C_DIS
LIN {X 0.258,Y -594.330,Z 1302.982,A 0.000,B 0.000,C 90.000,E1 32.673} C_DIS
LIN {X -0.348,Y -591.608,Z 1302.976,A 0.000,B 0.000,C 90.000,E1 31.671} C_DIS
LIN {X -0.063,Y -589.239,Z 1302.971,A 0.000,B 0.000,C 90.000,E1 30.846} C_DIS
LIN {X -0.290,Y -587.444,Z 1302.968,A 0.000,B 0.000,C 90.000,E1 30.335} C_DIS
LIN {X -0.229,Y -585.517,Z 1302.965,A 0.000,B 0.000,C 90.000,E1 29.795} C_DIS
LIN {X 0.323,Y -583.395,Z 1302.963,A 0.000,B 0.000,C 90.000,E1 29.205} C_DIS
LIN {X -0.064,Y -579.802,Z 1302.958,A 0.000,B 0.000,C 90.000,E1 28.437} C_DIS
LIN {X 0.004,Y -577.843,Z 1302.956,A 0.000,B 0.000,C 90.000,E1 28.025} C_DIS
LIN {X -0.004,Y -572.821,Z 1302.950,A 0.000,B 0.000,C 90.000,E1 27.078} C_DIS
LIN {X -0.154,Y -568.937,Z 1302.947,A 0.000,B 0.000,C 90.000,E1 26.411} C_DIS
LIN {X -0.082,Y -564.546,Z 1302.943,A 0.000,B 0.000,C 90.000,E1 25.720} C_DIS
LIN {X -0.047,Y -559.896,Z 1302.939,A 0.000,B 0.000,C 90.000,E1 25.027} C_DIS
LIN {X 0.054,Y -555.908,Z 1302.936,A 0.000,B 0.000,C 90.000,E1 24.463} C_DIS
LIN {X 0.015,Y -550.504,Z 1302.932,A 0.000,B 0.000,C 90.000,E1 23.770} C_DIS
LIN {X -0.076,Y -544.697,Z 1302.928,A 0.000,B 0.000,C 90.000,E1 23.078} C_DIS
LIN {X 0.025,Y -536.049,Z 1302.923,A 0.000,B 0.000,C 90.000,E1 22.078} C_DIS
LIN {X -0.088,Y -530.982,Z 1302.920,A 0.000,B 0.000,C 90.000,E1 21.535} C_DIS
LIN {X -0.042,Y -521.842,Z 1302.914,A 0.000,B 0.000,C 90.000,E1 20.556} C_DIS
LIN {X 0.154,Y -511.390,Z 1302.908,A 0.000,B 0.000,C 90.000,E1 19.450} C_DIS
LIN {X 0.050,Y -502.225,Z 1302.903,A 0.000,B 0.000,C 90.000,E1 18.544} C_DIS
LIN {X -0.091,Y -494.128,Z 1302.899,A 0.000,B 0.000,C 90.000,E1 17.764} C_DIS
LIN {X 0.184,Y -484.459,Z 1302.894,A 0.000,B 0.000,C 90.000,E1 16.804} C_DIS
LIN {X -0.057,Y -474.192,Z 1302.888,A 0.000,B 0.000,C 90.000,E1 15.898} C_DIS
LIN {X -0.183,Y -459.571,Z 1302.881,A 0.000,B 0.000,C 90.000,E1 14.592} C_DIS
LIN {X -0.182,Y -439.170,Z 1302.870,A 0.000,B 0.000,C 90.000,E1 12.647} C_DIS
LIN {X 0.054,Y -420.772,Z 1302.860,A 0.000,B 0.000,C 90.000,E1 10.715} C_DIS
LIN {X 0.074,Y -406.472,Z 1302.851,A 0.000,B 0.000,C 90.000,E1 9.151} C_DIS
LIN {X -0.023,Y -398.229,Z 1302.846,A 0.000,B 0.000,C 90.000,E1 8.219} C_DIS
LIN {X 0.057,Y -397.040,Z 1302.845,A 0.000,B 0.000,C 90.000,E1 8.049} C_DIS
LIN {X -0.041,Y -395.338,Z 1302.843,A 0.000,B 0.000,C 90.000,E1 7.757} C_DIS
LIN {X -0.079,Y -395.337,Z 1302.843,A 0.000,B 0.000,C 90.000,E1 7.757} C_DIS
LIN {X -0.130,Y -396.010,Z 1302.842,A 0.000,B 0.000,C 90.000,E1 7.644} C_DIS
LIN {X 0.082,Y -400.066,Z 1302.840,A 0.000,B 0.000,C 90.000,E1 7.239} C_DIS
LIN {X -0.084,Y -406.045,Z 1302.838,A 0.000,B 0.000,C 90.000,E1 6.891} C_DIS
LIN {X 0.160,Y -412.253,Z 1302.836,A 0.000,B 0.000,C 90.000,E1 6.486} C_DIS
LIN {X -0.073,Y -417.210,Z 1302.834,A 0.000,B 0.000,C 90.000,E1 6.201} C_DIS
LIN {X -0.114,Y -428.319,Z 1302.830,A 0.000,B 0.000,C 90.000,E1 5.391} C_DIS
LIN {X 0.037,Y -436.064,Z 1302.827,A 0.000,B 0.000,C 90.000,E1 4.759} C_DIS
LIN {X 0.154,Y -442.004,Z 1302.824,A 0.000,B 0.000,C 90.000,E1 4.245} C_DIS
LIN {X -0.139,Y -449.409,Z 1302.820,A 0.000,B 0.000,C 90.000,E1 3.612} C_DIS
LIN {X 0.037,Y -455.301,Z 1302.817,A 0.000,B 0.000,C 90.000,E1 3.037} C_DIS
LIN {X 0.113,Y -461.090,Z 1302.814,A 0.000,B 0.000,C 90.000,E1 2.465} C_DIS
LIN {X 0.207,Y -467.897,Z 1302.810,A 0.000,B 0.000,C 90.000,E1 1.718} C_DIS
LIN {X -0.209,Y -472.947,Z 1302.807,A 0.000,B 0.000,C 90.000,E1 1.203} C_DIS
LIN {X 0.160,Y -480.263,Z 1302.801,A 0.000,B 0.000,C 90.000,E1 0.229} C_DIS
LIN {X 0.152,Y -486.798,Z 1302.796,A 0.000,B 0.000,C 90.000,E1 359.312} C_DIS
LIN {X -0.188,Y -490.934,Z 1302.793,A 0.000,B 0.000,C 90.000,E1 358.740} C_DIS
LIN {X -0.142,Y -496.455,Z 1302.788,A 0.000,B 0.000,C 90.000,E1 357.822} C_DIS
LIN {X -0.051,Y -501.577,Z 1302.783,A 0.000,B 0.000,C 90.000,E1 356.906} C_DIS
LIN {X 0.235,Y -504.780,Z 1302.780,A 0.000,B 0.000,C 90.000,E1 356.274} C_DIS
LIN {X 0.141,Y -510.046,Z 1302.774,A 0.000,B 0.000,C 90.000,E1 355.241} C_DIS
LIN {X 0.156,Y -514.730,Z 1302.768,A 0.000,B 0.000,C 90.000,E1 354.204} C_DIS
LIN {X 0.234,Y -519.137,Z 1302.762,A 0.000,B 0.000,C 90.000,E1 353.166} C_DIS
LIN {X 0.137,Y -523.449,Z 1302.756,A 0.000,B 0.000,C 90.000,E1 352.008} C_DIS
LIN {X 0.087,Y -526.443,Z 1302.751,A 0.000,B 0.000,C 90.000,E1 351.141} C_DIS
LIN {X 0.091,Y -529.941,Z 1302.745,A 0.000,B 0.000,C 90.000,E1 349.982} C_DIS
LIN {X 0.196,Y -532.288,Z 1302.740,A 0.000,B 0.000,C 90.000,E1 349.106} C_DIS
LIN {X -0.241,Y -533.762,Z 1302.736,A 0.000,B 0.000,C 90.000,E1 348.578} C_DIS
LIN {X -0.038,Y -536.292,Z 1302.730,A 0.000,B 0.000,C 90.000,E1 347.409} C_DIS
LIN {X -0.201,Y -538.465,Z 1302.724,A 0.000,B 0.000,C 90.000,E1 346.284} C_DIS
LIN {X -0.008,Y -539.861,Z 1302.719,A 0.000,B 0.000,C 90.000,E1 345.408} C_DIS
LIN {X -0.191,Y -540.997,Z 1302.714,A 0.000,B 0.000,C 90.000,E1 344.574} C_DIS
LIN {X 0.160,Y -541.850,Z 1302.709,A 0.000,B 0.000,C 90.000,E1 343.685} C_DIS
LIN {X -0.004,Y -542.495,Z 1302.705,A 0.000,B 0.000,C 90.000,E1 342.851} C_DIS
LIN {X 0.065,Y -542.960,Z 1302.698,A 0.000,B 0.000,C 90.000,E1 341.710} C_DIS
LIN {X 0.019,Y -543.028,Z 1302.695,A 0.000,B 0.000,C 90.000,E1 341.148} C_DIS
LIN {X 0.041,Y -542.740,Z 1302.691,A 0.000,B 0.000,C 90.000,E1 340.296} C_DIS
LIN {X 0.060,Y -542.276,Z 1302.686,A 0.000,B 0.000,C 90.000,E1 339.444} C_DIS
LIN {X -0.165,Y -541.846,Z 1302.683,A 0.000,B 0.000,C 90.000,E1 338.901} C_DIS
LIN {X -0.207,Y -539.893,Z 1302.675,A 0.000,B 0.000,C 90.000,E1 337.486} C_DIS
LIN {X -0.250,Y -539.018,Z 1302.672,A 0.000,B 0.000,C 90.000,E1 336.922} C_DIS
LIN {X -0.026,Y -538.493,Z 1302.670,A 0.000,B 0.000,C 90.000,E1 336.613} C_DIS
LIN {X 0.196,Y -537.760,Z 1302.669,A 0.000,B 0.000,C 90.000,E1 336.305} C_DIS
LIN {X 0.137,Y -536.568,Z 1302.665,A 0.000,B 0.000,C 90.000,E1 335.741} C_DIS
LIN {X -0.210,Y -534.201,Z 1302.661,A 0.000,B 0.000,C 90.000,E1 334.921} C_DIS
LIN {X 0.130,Y -531.605,Z 1302.656,A 0.000,B 0.000,C 90.000,E1 334.024} C_DIS
LIN {X -0.156,Y -526.923,Z 1302.648,A 0.000,B 0.000,C 90.000,E1 332.615} C_DIS
LIN {X 0.037,Y -522.837,Z 1302.641,A 0.000,B 0.000,C 90.000,E1 331.435} C_DIS
LIN {X 0.170,Y -518.353,Z 1302.635,A 0.000,B 0.000,C 90.000,E1 330.255} C_DIS
LIN {X -0.133,Y -514.562,Z 1302.630,A 0.000,B 0.000,C 90.000,E1 329.410} C_DIS
LIN {X -0.064,Y -508.457,Z 1302.623,A 0.000,B 0.000,C 90.000,E1 328.074} C_DIS
LIN {X -0.028,Y -501.641,Z 1302.614,A 0.000,B 0.000,C 90.000,E1 326.580} C_DIS
LIN {X -0.175,Y -499.047,Z 1302.610,A 0.000,B 0.000,C 90.000,E1 325.881} C_DIS
LIN {X 0.010,Y -497.446,Z 1302.607,A 0.000,B 0.000,C 90.000,E1 325.261} C_DIS
LIN {X -0.254,Y -496.080,Z 1302.604,A 0.000,B 0.000,C 90.000,E1 324.689} C_DIS
LIN {X 0.030,Y -494.666,Z 1302.599,A 0.000,B 0.000,C 90.000,E1 323.749} C_DIS
LIN {X -0.284,Y -493.375,Z 1302.590,A 0.000,B 0.000,C 90.000,E1 322.271} C_DIS
LIN {X -0.021,Y -492.809,Z 1302.582,A 0.000,B 0.000,C 90.000,E1 320.723} C_DIS
LIN {X -0.128,Y -492.870,Z 1302.570,A 0.000,B 0.000,C 90.000,E1 318.609} C_DIS
LIN {X 0.062,Y -492.651,Z 1302.565,A 0.000,B 0.000,C 90.000,E1 317.676} C_DIS
LIN {X 0.076,Y -492.194,Z 1302.562,A 0.000,B 0.000,C 90.000,E1 317.067} C_DIS
LIN {X 0.083,Y -491.432,Z 1302.558,A 0.000,B 0.000,C 90.000,E1 316.458} C_DIS
LIN {X 0.253,Y -490.887,Z 1302.557,A 0.000,B 0.000,C 90.000,E1 316.134} C_DIS
LIN {X -0.272,Y -490.176,Z 1302.555,A 0.000,B 0.000,C 90.000,E1 315.891} C_DIS
LIN {X -0.104,Y -489.184,Z 1302.553,A 0.000,B 0.000,C 90.000,E1 315.567} C_DIS
LIN {X -0.021,Y -488.475,Z 1302.552,A 0.000,B 0.000,C 90.000,E1 315.405} C_DIS
LIN {X 0.061,Y -487.404,Z 1302.551,A 0.000,B 0.000,C 90.000,E1 315.243} C_DIS
LIN {X 0.079,Y -467.189,Z 1302.538,A 0.000,B 0.000,C 90.000,E1 312.771} C_DIS
LIN {X -0.170,Y -448.840,Z 1302.524,A 0.000,B 0.000,C 90.000,E1 310.253} C_DIS
LIN {X 0.068,Y -432.285,Z 1302.509,A 0.000,B 0.000,C 90.000,E1 307.604} C_DIS
LIN {X -0.130,Y -417.405,Z 1302.494,A 0.000,B 0.000,C 90.000,E1 304.945} C_DIS
LIN {X -0.226,Y -404.096,Z 1302.479,A 0.000,B 0.000,C 90.000,E1 302.212} C_DIS
LIN {X 0.051,Y -395.111,Z 1302.467,A 0.000,B 0.000,C 90.000,E1 300.079} C_DIS
LIN {X 0.013,Y -395.110,Z 1302.467,A 0.000,B 0.000,C 90.000,E1 300.079} C_DIS
LIN {X 0.015,Y -397.043,Z 1302.458,A 0.000,B 0.000,C 90.000,E1 298.487} C_DIS
LIN {X -0.205,Y -401.425,Z 1302.427,A 0.000,B 0.000,C 90.000,E1 292.898} C_DIS
LIN {X 0.031,Y -401.671,Z 1302.425,A 0.000,B 0.000,C 90.000,E1 292.514} C_DIS
LIN {X 0.162,Y -404.763,Z 1302.394,A 0.000,B 0.000,C 90.000,E1 286.913} C_DIS
LIN {X 0.069,Y -406.155,Z 1302.363,A 0.000,B 0.000,C 90.000,E1 281.366} C_DIS
LIN {X 0.173,Y -405.643,Z 1302.334,A 0.000,B 0.000,C 90.000,E1 276.144} C_DIS
LIN {X 0.178,Y -405.641,Z 1302.332,A 0.000,B 0.000,C 90.000,E1 275.796} C_DIS
LIN {X -0.152,Y -403.557,Z 1302.305,A 0.000,B 0.000,C 90.000,E1 270.974} C_DIS
LIN {X 0.186,Y -403.100,Z 1302.302,A 0.000,B 0.000,C 90.000,E1 270.229} C_DIS
LIN {X 0.011,Y -399.034,Z 1302.272,A 0.000,B 0.000,C 90.000,E1 265.008} C_DIS
LIN {X -0.048,Y -398.672,Z 1302.270,A 0.000,B 0.000,C 90.000,E1 264.666} C_DIS
LIN {X -0.165,Y -393.233,Z 1302.243,A 0.000,B 0.000,C 90.000,E1 259.746} C_DIS
LIN {X -0.204,Y -392.964,Z 1302.241,A 0.000,B 0.000,C 90.000,E1 259.398} C_DIS
LIN {X 0.140,Y -392.547,Z 1302.239,A 0.000,B 0.000,C 90.000,E1 258.993} C_DIS
LIN {X -0.085,Y -386.167,Z 1302.213,A 0.000,B 0.000,C 90.000,E1 254.393} C_DIS
LIN {X -0.122,Y -385.056,Z 1302.207,A 0.000,B 0.000,C 90.000,E1 253.323} C_DIS
LIN {X 0.118,Y -378.187,Z 1302.183,A 0.000,B 0.000,C 90.000,E1 248.954} C_DIS
LIN {X -0.161,Y -375.961,Z 1302.173,A 0.000,B 0.000,C 90.000,E1 247.177} C_DIS
LIN {X -0.115,Y -374.184,Z 1302.168,A 0.000,B 0.000,C 90.000,E1 246.230} C_DIS
LIN {X -0.152,Y -374.187,Z 1302.168,A 0.000,B 0.000,C 90.000,E1 246.230} C_DIS
LIN {X 0.134,Y -384.070,Z 1302.151,A 0.000,B 0.000,C 90.000,E1 243.127} C_DIS
LIN {X -0.118,Y -395.567,Z 1302.134,A 0.000,B 0.000,C 90.000,E1 240.127} C_DIS
LIN {X -0.140,Y -407.858,Z 1302.118,A 0.000,B 0.000,C 90.000,E1 237.327} C_DIS
LIN {X 0.001,Y -421.664,Z 1302.103,A 0.000,B 0.000,C 90.000,E1 234.562} C_DIS
LIN {X -0.180,Y -437.085,Z 1302.088,A 0.000,B 0.000,C 90.000,E1 231.904} C_DIS
LIN {X 0.040,Y -448.682,Z 1302.078,A 0.000,B 0.000,C 90.000,E1 230.070} C_DIS
LIN {X 0.032,Y -449.523,Z 1302.077,A 0.000,B 0.000,C 90.000,E1 229.908} C_DIS
LIN {X 0.025,Y -450.105,Z 1302.076,A 0.000,B 0.000,C 90.000,E1 229.747} C_DIS
LIN {X -0.273,Y -450.927,Z 1302.075,A 0.000,B 0.000,C 90.000,E1 229.461} C_DIS
LIN {X 0.066,Y -451.505,Z 1302.073,A 0.000,B 0.000,C 90.000,E1 229.094} C_DIS
LIN {X 0.073,Y -452.255,Z 1302.069,A 0.000,B 0.000,C 90.000,E1 228.447} C_DIS
LIN {X 0.125,Y -452.636,Z 1302.066,A 0.000,B 0.000,C 90.000,E1 227.796} C_DIS
LIN {X -0.148,Y -452.873,Z 1302.060,A 0.000,B 0.000,C 90.000,E1 226.863} C_DIS
LIN {X -0.090,Y -452.761,Z 1302.053,A 0.000,B 0.000,C 90.000,E1 225.567} C_DIS
LIN {X -0.002,Y -452.638,Z 1302.042,A 0.000,B 0.000,C 90.000,E1 223.623} C_DIS
LIN {X 0.038,Y -453.985,Z 1302.016,A 0.000,B 0.000,C 90.000,E1 218.785} C_DIS
LIN {X 0.207,Y -455.127,Z 1302.007,A 0.000,B 0.000,C 90.000,E1 217.156} C_DIS
LIN {X -0.069,Y -456.877,Z 1301.994,A 0.000,B 0.000,C 90.000,E1 214.945} C_DIS
LIN {X -0.088,Y -459.953,Z 1301.976,A 0.000,B 0.000,C 90.000,E1 211.750} C_DIS
LIN {X 0.035,Y -463.453,Z 1301.960,A 0.000,B 0.000,C 90.000,E1 208.871} C_DIS
LIN {X -0.002,Y -467.291,Z 1301.945,A 0.000,B 0.000,C 90.000,E1 206.027} C_DIS
LIN {X 0.051,Y -470.048,Z 1301.934,A 0.000,B 0.000,C 90.000,E1 204.131} C_DIS
LIN {X -0.167,Y -472.306,Z 1301.925,A 0.000,B 0.000,C 90.000,E1 202.589} C_DIS
LIN {X 0.052,Y -475.433,Z 1301.913,A 0.000,B 0.000,C 90.000,E1 200.375} C_DIS
LIN {X -0.245,Y -478.389,Z 1301.903,A 0.000,B 0.000,C 90.000,E1 198.544} C_DIS
LIN {X -0.183,Y -481.245,Z 1301.893,A 0.000,B 0.000,C 90.000,E1 196.677} C_DIS
LIN {X -0.199,Y -484.119,Z 1301.882,A 0.000,B 0.000,C 90.000,E1 194.828} C_DIS
LIN {X 0.192,Y -487.027,Z 1301.872,A 0.000,B 0.000,C 90.000,E1 192.939} C_DIS
LIN {X -0.150,Y -490.270,Z 1301.860,A 0.000,B 0.000,C 90.000,E1 190.838} C_DIS
LIN {X 0.179,Y -493.023,Z 1301.850,A 0.000,B 0.000,C 90.000,E1 188.973} C_DIS
LIN {X 0.026,Y -495.306,Z 1301.842,A 0.000,B 0.000,C 90.000,E1 187.473} C_DIS
LIN {X -0.023,Y -497.557,Z 1301.833,A 0.000,B 0.000,C 90.000,E1 185.967} C_DIS
LIN {X -0.142,Y -499.714,Z 1301.825,A 0.000,B 0.000,C 90.000,E1 184.473} C_DIS
LIN {X 0.158,Y -502.073,Z 1301.815,A 0.000,B 0.000,C 90.000,E1 182.636} C_DIS
LIN {X -0.178,Y -503.124,Z 1301.810,A 0.000,B 0.000,C 90.000,E1 181.776} C_DIS
LIN {X -0.236,Y -504.698,Z 1301.802,A 0.000,B 0.000,C 90.000,E1 180.286} C_DIS
LIN {X -0.157,Y -505.859,Z 1301.795,A 0.000,B 0.000,C 90.000,E1 179.083} C_DIS
LIN {X 0.052,Y -506.556,Z 1301.790,A 0.000,B 0.000,C 90.000,E1 178.165} C_DIS
LIN {X 0.077,Y -507.471,Z 1301.782,A 0.000,B 0.000,C 90.000,E1 176.674} C_DIS
LIN {X 0.209,Y -507.978,Z 1301.775,A 0.000,B 0.000,C 90.000,E1 175.469} C_DIS
LIN {X -0.122,Y -508.155,Z 1301.768,A 0.000,B 0.000,C 90.000,E1 174.318} C_DIS
LIN {X 0.055,Y -508.032,Z 1301.762,A 0.000,B 0.000,C 90.000,E1 173.109} C_DIS
LIN {X -0.164,Y -507.844,Z 1301.757,A 0.000,B 0.000,C 90.000,E1 172.243} C_DIS
LIN {X 0.115,Y -507.304,Z 1301.752,A 0.000,B 0.000,C 90.000,E1 171.319} C_DIS
LIN {X -0.034,Y -506.515,Z 1301.747,A 0.000,B 0.000,C 90.000,E1 170.443} C_DIS
LIN {X 0.261,Y -505.146,Z 1301.740,A 0.000,B 0.000,C 90.000,E1 169.218} C_DIS
LIN {X 0.099,Y -503.852,Z 1301.735,A 0.000,B 0.000,C 90.000,E1 168.342} C_DIS
LIN {X -0.079,Y -502.194,Z 1301.730,A 0.000,B 0.000,C 90.000,E1 167.465} C_DIS
LIN {X -0.278,Y -500.381,Z 1301.725,A 0.000,B 0.000,C 90.000,E1 166.589} C_DIS
LIN {X 0.100,Y -498.238,Z 1301.720,A 0.000,B 0.000,C 90.000,E1 165.644} C_DIS
LIN {X -0.027,Y -495.936,Z 1301.715,A 0.000,B 0.000,C 90.000,E1 164.755} C_DIS
LIN {X -0.146,Y -492.823,Z 1301.709,A 0.000,B 0.000,C 90.000,E1 163.559} C_DIS
LIN {X 0.157,Y -489.419,Z 1301.702,A 0.000,B 0.000,C 90.000,E1 162.308} C_DIS
LIN {X -0.136,Y -483.964,Z 1301.694,A 0.000,B 0.000,C 90.000,E1 160.967} C_DIS
LIN {X -0.060,Y -478.498,Z 1301.687,A 0.000,B 0.000,C 90.000,E1 159.571} C_DIS
LIN {X -0.081,Y -476.562,Z 1301.683,A 0.000,B 0.000,C 90.000,E1 158.954} C_DIS
LIN {X -0.115,Y -475.113,Z 1301.680,A 0.000,B 0.000,C 90.000,E1 158.337} C_DIS
LIN {X -0.137,Y -474.880,Z 1301.678,A 0.000,B 0.000,C 90.000,E1 158.028} C_DIS
LIN {X -0.187,Y -475.021,Z 1301.674,A 0.000,B 0.000,C 90.000,E1 157.411} C_DIS
LIN {X 0.052,Y -476.242,Z 1301.672,A 0.000,B 0.000,C 90.000,E1 156.975} C_DIS
LIN {X 0.011,Y -476.281,Z 1301.672,A 0.000,B 0.000,C 90.000,E1 156.975} C_DIS
LIN {X 0.038,Y -477.067,Z 1301.672,A 0.000,B 0.000,C 90.000,E1 156.869} C_DIS
LIN {X -0.193,Y -478.025,Z 1301.671,A 0.000,B 0.000,C 90.000,E1 156.741} C_DIS
LIN {X -0.119,Y -479.013,Z 1301.670,A 0.000,B 0.000,C 90.000,E1 156.538} C_DIS
LIN {X 0.191,Y -481.833,Z 1301.668,A 0.000,B 0.000,C 90.000,E1 156.230} C_DIS
LIN {X 0.105,Y -482.980,Z 1301.667,A 0.000,B 0.000,C 90.000,E1 156.102} C_DIS
LIN {X -0.079,Y -494.334,Z 1301.662,A 0.000,B 0.000,C 90.000,E1 155.101} C_DIS
LIN {X -0.207,Y -500.009,Z 1301.659,A 0.000,B 0.000,C 90.000,E1 154.588} C_DIS
LIN {X 0.117,Y -505.300,Z 1301.656,A 0.000,B 0.000,C 90.000,E1 154.024} C_DIS
LIN {X 0.088,Y -510.526,Z 1301.653,A 0.000,B 0.000,C 90.000,E1 153.461} C_DIS
LIN {X -0.166,Y -514.392,Z 1301.650,A 0.000,B 0.000,C 90.000,E1 153.050} C_DIS
LIN {X 0.082,Y -519.109,Z 1301.647,A 0.000,B 0.000,C 90.000,E1 152.436} C_DIS
LIN {X 0.121,Y -523.299,Z 1301.644,A 0.000,B 0.000,C 90.000,E1 151.847} C_DIS
LIN {X 0.193,Y -527.015,Z 1301.641,A 0.000,B 0.000,C 90.000,E1 151.257} C_DIS
LIN {X 0.141,Y -530.845,Z 1301.636,A 0.000,B 0.000,C 90.000,E1 150.539} C_DIS
LIN {X -0.193,Y -533.312,Z 1301.633,A 0.000,B 0.000,C 90.000,E1 149.999} C_DIS
LIN {X -0.049,Y -535.367,Z 1301.630,A 0.000,B 0.000,C 90.000,E1 149.410} C_DIS
LIN {X 0.107,Y -537.125,Z 1301.627,A 0.000,B 0.000,C 90.000,E1 148.820} C_DIS
LIN {X 0.100,Y -537.939,Z 1301.625,A 0.000,B 0.000,C 90.000,E1 148.535} C_DIS
LIN {X -0.005,Y -540.685,Z 1301.619,A 0.000,B 0.000,C 90.000,E1 147.406} C_DIS
LIN {X -0.036,Y -541.916,Z 1301.618,A 0.000,B 0.000,C 90.000,E1 147.199} C_DIS
LIN {X 0.118,Y -542.563,Z 1301.617,A 0.000,B 0.000,C 90.000,E1 147.041} C_DIS
LIN {X 0.141,Y -543.461,Z 1301.615,A 0.000,B 0.000,C 90.000,E1 146.755} C_DIS
LIN {X 0.004,Y -544.811,Z 1301.615,A 0.000,B 0.000,C 90.000,E1 146.628} C_DIS
LIN {X 0.087,Y -545.904,Z 1301.614,A 0.000,B 0.000,C 90.000,E1 146.548} C_DIS
LIN {X -0.164,Y -557.171,Z 1301.611,A 0.000,B 0.000,C 90.000,E1 146.008} C_DIS
LIN {X -0.060,Y -566.431,Z 1301.608,A 0.000,B 0.000,C 90.000,E1 145.468} C_DIS
LIN {X 0.181,Y -572.421,Z 1301.606,A 0.000,B 0.000,C 90.000,E1 145.055} C_DIS
LIN {X -0.353,Y -581.328,Z 1301.603,A 0.000,B 0.000,C 90.000,E1 144.482} C_DIS
LIN {X -0.176,Y -588.331,Z 1301.599,A 0.000,B 0.000,C 90.000,E1 143.909} C_DIS
LIN {X -0.065,Y -589.761,Z 1301.599,A 0.000,B 0.000,C 90.000,E1 143.783} C_DIS
LIN {X -0.008,Y -596.066,Z 1301.595,A 0.000,B 0.000,C 90.000,E1 143.176} C_DIS
LIN {X 0.012,Y -599.744,Z 1301.593,A 0.000,B 0.000,C 90.000,E1 142.798} C_DIS
LIN {X 0.033,Y -604.444,Z 1301.590,A 0.000,B 0.000,C 90.000,E1 142.271} C_DIS
LIN {X -0.241,Y -607.736,Z 1301.588,A 0.000,B 0.000,C 90.000,E1 141.904} C_DIS
LIN {X -0.173,Y -611.768,Z 1301.585,A 0.000,B 0.000,C 90.000,E1 141.376} C_DIS
LIN {X -0.119,Y -616.376,Z 1301.582,A 0.000,B 0.000,C 90.000,E1 140.723} C_DIS
LIN {X -0.336,Y -619.016,Z 1301.580,A 0.000,B 0.000,C 90.000,E1 140.356} C_DIS
LIN {X 0.176,Y -623.023,Z 1301.576,A 0.000,B 0.000,C 90.000,E1 139.666} C_DIS
LIN {X -0.189,Y -627.455,Z 1301.572,A 0.000,B 0.000,C 90.000,E1 138.933} C_DIS
LIN {X -0.065,Y -630.994,Z 1301.568,A 0.000,B 0.000,C 90.000,E1 138.286} C_DIS
LIN {X -0.107,Y -637.270,Z 1301.561,A 0.000,B 0.000,C 90.000,E1 137.025} C_DIS
LIN {X 0.017,Y -641.441,Z 1301.556,A 0.000,B 0.000,C 90.000,E1 136.134} C_DIS
LIN {X -0.296,Y -646.082,Z 1301.551,A 0.000,B 0.000,C 90.000,E1 135.162} C_DIS
LIN {X 0.312,Y -651.648,Z 1301.544,A 0.000,B 0.000,C 90.000,E1 133.866} C_DIS
LIN {X -0.363,Y -657.121,Z 1301.537,A 0.000,B 0.000,C 90.000,E1 132.690} C_DIS
LIN {X -0.002,Y -661.453,Z 1301.532,A 0.000,B 0.000,C 90.000,E1 131.676} C_DIS
LIN {X -0.022,Y -665.550,Z 1301.526,A 0.000,B 0.000,C 90.000,E1 130.701} C_DIS
LIN {X 0.022,Y -668.499,Z 1301.522,A 0.000,B 0.000,C 90.000,E1 129.967} C_DIS
LIN {X -0.420,Y -671.292,Z 1301.518,A 0.000,B 0.000,C 90.000,E1 129.277} C_DIS
LIN {X 0.217,Y -675.618,Z 1301.511,A 0.000,B 0.000,C 90.000,E1 128.016} C_DIS
LIN {X -0.052,Y -678.038,Z 1301.507,A 0.000,B 0.000,C 90.000,E1 127.317} C_DIS
LIN {X 0.113,Y -680.261,Z 1301.503,A 0.000,B 0.000,C 90.000,E1 126.583} C_DIS
LIN {X -0.094,Y -683.045,Z 1301.498,A 0.000,B 0.000,C 90.000,E1 125.644} C_DIS
LIN {X -0.094,Y -686.173,Z 1301.491,A 0.000,B 0.000,C 90.000,E1 124.452} C_DIS
LIN {X 0.308,Y -687.876,Z 1301.487,A 0.000,B 0.000,C 90.000,E1 123.706} C_DIS
LIN {X 0.369,Y -689.838,Z 1301.482,A 0.000,B 0.000,C 90.000,E1 122.752} C_DIS
LIN {X 0.093,Y -691.913,Z 1301.476,A 0.000,B 0.000,C 90.000,E1 121.592} C_DIS
LIN {X 0.081,Y -693.702,Z 1301.469,A 0.000,B 0.000,C 90.000,E1 120.413} C_DIS
LIN {X 0.203,Y -695.068,Z 1301.464,A 0.000,B 0.000,C 90.000,E1 119.461} C_DIS
LIN {X 0.345,Y -695.878,Z 1301.460,A 0.000,B 0.000,C 90.000,E1 118.743} C_DIS
LIN {X -0.187,Y -696.743,Z 1301.455,A 0.000,B 0.000,C 90.000,E1 117.847} C_DIS
LIN {X -0.027,Y -697.104,Z 1301.451,A 0.000,B 0.000,C 90.000,E1 117.129} C_DIS
LIN {X 0.085,Y -697.239,Z 1301.446,A 0.000,B 0.000,C 90.000,E1 116.181} C_DIS
LIN {X 0.242,Y -696.997,Z 1301.442,A 0.000,B 0.000,C 90.000,E1 115.463} C_DIS
LIN {X -0.165,Y -696.610,Z 1301.439,A 0.000,B 0.000,C 90.000,E1 115.027} C_DIS
LIN {X 0.350,Y -695.901,Z 1301.436,A 0.000,B 0.000,C 90.000,E1 114.515} C_DIS
LIN {X -0.315,Y -695.488,Z 1301.435,A 0.000,B 0.000,C 90.000,E1 114.335} C_DIS
LIN {X 0.191,Y -693.954,Z 1301.432,A 0.000,B 0.000,C 90.000,E1 113.823} C_DIS
LIN {X 0.161,Y -692.945,Z 1301.431,A 0.000,B 0.000,C 90.000,E1 113.590} C_DIS
LIN {X 0.008,Y -689.921,Z 1301.429,A 0.000,B 0.000,C 90.000,E1 113.131} C_DIS
LIN {X -0.147,Y -688.914,Z 1301.428,A 0.000,B 0.000,C 90.000,E1 113.025} C_DIS
LIN {X -0.030,Y -687.395,Z 1301.427,A 0.000,B 0.000,C 90.000,E1 112.898} C_DIS
LIN {X -0.017,Y -682.891,Z 1301.426,A 0.000,B 0.000,C 90.000,E1 112.589} C_DIS
LIN {X -0.289,Y -681.316,Z 1301.425,A 0.000,B 0.000,C 90.000,E1 112.514} C_DIS
LIN {X 0.135,Y -678.922,Z 1301.424,A 0.000,B 0.000,C 90.000,E1 112.386} C_DIS
LIN {X -0.108,Y -672.548,Z 1301.423,A 0.000,B 0.000,C 90.000,E1 112.206} C_DIS
LIN {X 0.178,Y -667.354,Z 1301.423,A 0.000,B 0.000,C 90.000,E1 112.099} C_DIS
LIN {X -0.167,Y -663.283,Z 1301.423,A 0.000,B 0.000,C 90.000,E1 112.078} C_DIS
LIN {X 0.021,Y -656.041,Z 1301.422,A 0.000,B 0.000,C 90.000,E1 112.025} C_DIS
LIN {X -0.126,Y -649.435,Z 1301.422,A 0.000,B 0.000,C 90.000,E1 112.025} C_DIS
LIN {X -0.113,Y -644.367,Z 1301.422,A 0.000,B 0.000,C 90.000,E1 111.972} C_DIS
LIN {X 0.192,Y -640.886,Z 1301.422,A 0.000,B 0.000,C 90.000,E1 111.844} C_DIS
LIN {X 0.152,Y -640.833,Z 1301.422,A 0.000,B 0.000,C 90.000,E1 111.844} C_DIS
LIN {X -0.158,Y -642.513,Z 1301.420,A 0.000,B 0.000,C 90.000,E1 111.535} C_DIS
LIN {X 0.131,Y -650.884,Z 1301.414,A 0.000,B 0.000,C 90.000,E1 110.429} C_DIS
LIN {X 0.111,Y -655.029,Z 1301.410,A 0.000,B 0.000,C 90.000,E1 109.812} C_DIS
LIN {X -0.094,Y -658.591,Z 1301.407,A 0.000,B 0.000,C 90.000,E1 109.214} C_DIS
LIN {X -0.056,Y -661.801,Z 1301.403,A 0.000,B 0.000,C 90.000,E1 108.598} C_DIS
LIN {X -0.153,Y -665.101,Z 1301.399,A 0.000,B 0.000,C 90.000,E1 107.873} C_DIS
LIN {X -0.335,Y -667.107,Z 1301.397,A 0.000,B 0.000,C 90.000,E1 107.402} C_DIS
LIN {X 0.258,Y -669.668,Z 1301.393,A 0.000,B 0.000,C 90.000,E1 106.622} C_DIS
LIN {X 0.114,Y -671.177,Z 1301.390,A 0.000,B 0.000,C 90.000,E1 106.150} C_DIS
LIN {X 0.040,Y -673.636,Z 1301.384,A 0.000,B 0.000,C 90.000,E1 105.190} C_DIS
LIN {X -0.075,Y -674.669,Z 1301.382,A 0.000,B 0.000,C 90.000,E1 104.717} C_DIS
LIN {X -0.285,Y -676.382,Z 1301.376,A 0.000,B 0.000,C 90.000,E1 103.772} C_DIS
LIN {X 0.232,Y -677.156,Z 1301.372,A 0.000,B 0.000,C 90.000,E1 103.008} C_DIS
LIN {X 0.094,Y -677.614,Z 1301.368,A 0.000,B 0.000,C 90.000,E1 102.299} C_DIS
LIN {X 0.048,Y -677.740,Z 1301.367,A 0.000,B 0.000,C 90.000,E1 102.063} C_DIS
LIN {X -0.227,Y -677.637,Z 1301.363,A 0.000,B 0.000,C 90.000,E1 101.366} C_DIS
LIN {X -0.321,Y -677.373,Z 1301.360,A 0.000,B 0.000,C 90.000,E1 100.894} C_DIS
LIN {X 0.244,Y -676.927,Z 1301.358,A 0.000,B 0.000,C 90.000,E1 100.366} C_DIS
LIN {X -0.036,Y -675.750,Z 1301.354,A 0.000,B 0.000,C 90.000,E1 99.670} C_DIS
LIN {X -0.263,Y -674.673,Z 1301.351,A 0.000,B 0.000,C 90.000,E1 99.208} C_DIS
LIN {X 0.173,Y -673.283,Z 1301.348,A 0.000,B 0.000,C 90.000,E1 98.690} C_DIS
LIN {X 0.033,Y -671.472,Z 1301.346,A 0.000,B 0.000,C 90.000,E1 98.219} C_DIS
LIN {X -0.215,Y -669.306,Z 1301.343,A 0.000,B 0.000,C 90.000,E1 97.757} C_DIS
LIN {X 0.099,Y -666.379,Z 1301.340,A 0.000,B 0.000,C 90.000,E1 97.125} C_DIS
LIN {X -0.289,Y -662.249,Z 1301.336,A 0.000,B 0.000,C 90.000,E1 96.429} C_DIS
LIN {X 0.060,Y -659.292,Z 1301.333,A 0.000,B 0.000,C 90.000,E1 95.910} C_DIS
LIN {X -0.267,Y -656.005,Z 1301.330,A 0.000,B 0.000,C 90.000,E1 95.448} C_DIS
LIN {X -0.030,Y -651.507,Z 1301.327,A 0.000,B 0.000,C 90.000,E1 94.821} C_DIS
LIN {X 0.243,Y -647.522,Z 1301.324,A 0.000,B 0.000,C 90.000,E1 94.302} C_DIS
LIN {X 0.249,Y -640.831,Z 1301.320,A 0.000,B 0.000,C 90.000,E1 93.555} C_DIS
LIN {X -0.305,Y -634.976,Z 1301.316,A 0.000,B 0.000,C 90.000,E1 92.980} C_DIS
LIN {X 0.237,Y -627.755,Z 1301.312,A 0.000,B 0.000,C 90.000,E1 92.178} C_DIS
LIN {X -0.127,Y -622.677,Z 1301.310,A 0.000,B 0.000,C 90.000,E1 91.718} C_DIS
LIN {X -0.201,Y -615.815,Z 1301.306,A 0.000,B 0.000,C 90.000,E1 91.146} C_DIS
LIN {X 0.002,Y -609.684,Z 1301.304,A 0.000,B 0.000,C 90.000,E1 90.688} C_DIS
LIN {X 0.269,Y -601.876,Z 1301.301,A 0.000,B 0.000,C 90.000,E1 90.172} C_DIS
LIN {X 0.197,Y -595.345,Z 1301.299,A 0.000,B 0.000,C 90.000,E1 89.828} C_DIS
LIN {X -0.104,Y -588.375,Z 1301.297,A 0.000,B 0.000,C 90.000,E1 89.542} C_DIS
LIN {X 0.021,Y -576.243,Z 1301.295,A 0.000,B 0.000,C 90.000,E1 89.083} C_DIS
LIN {X 0.067,Y -572.514,Z 1301.294,A 0.000,B 0.000,C 90.000,E1 88.912} C_DIS
LIN {X -0.109,Y -571.205,Z 1301.294,A 0.000,B 0.000,C 90.000,E1 88.854} C_DIS
LIN {X -0.281,Y -570.701,Z 1301.293,A 0.000,B 0.000,C 90.000,E1 88.797} C_DIS
LIN {X -0.136,Y -570.036,Z 1301.292,A 0.000,B 0.000,C 90.000,E1 88.625} C_DIS
LIN {X -0.149,Y -569.952,Z 1301.290,A 0.000,B 0.000,C 90.000,E1 88.165} C_DIS
LIN {X -0.230,Y -571.733,Z 1301.278,A 0.000,B 0.000,C 90.000,E1 85.988} C_DIS
LIN {X -0.145,Y -574.064,Z 1301.266,A 0.000,B 0.000,C 90.000,E1 83.799} C_DIS
LIN {X 0.126,Y -575.649,Z 1301.258,A 0.000,B 0.000,C 90.000,E1 82.413} C_DIS
LIN {X -0.177,Y -578.261,Z 1301.246,A 0.000,B 0.000,C 90.000,E1 80.274} C_DIS
LIN {X 0.128,Y -579.510,Z 1301.240,A 0.000,B 0.000,C 90.000,E1 79.162} C_DIS
LIN {X -0.003,Y -580.808,Z 1301.232,A 0.000,B 0.000,C 90.000,E1 77.825} C_DIS
LIN {X 0.134,Y -582.043,Z 1301.225,A 0.000,B 0.000,C 90.000,E1 76.464} C_DIS
LIN {X 0.156,Y -583.056,Z 1301.217,A 0.000,B 0.000,C 90.000,E1 75.117} C_DIS
LIN {X -0.070,Y -584.006,Z 1301.210,A 0.000,B 0.000,C 90.000,E1 73.795} C_DIS
LIN {X -0.038,Y -585.039,Z 1301.201,A 0.000,B 0.000,C 90.000,E1 72.181} C_DIS
LIN {X -0.222,Y -585.955,Z 1301.194,A 0.000,B 0.000,C 90.000,E1 70.859} C_DIS
LIN {X 0.217,Y -586.937,Z 1301.185,A 0.000,B 0.000,C 90.000,E1 69.209} C_DIS
LIN {X 0.004,Y -588.087,Z 1301.174,A 0.000,B 0.000,C 90.000,E1 67.358} C_DIS
LIN {X 0.158,Y -589.187,Z 1301.165,A 0.000,B 0.000,C 90.000,E1 65.741} C_DIS
LIN {X -0.065,Y -590.478,Z 1301.155,A 0.000,B 0.000,C 90.000,E1 63.896} C_DIS
LIN {X -0.087,Y -592.248,Z 1301.143,A 0.000,B 0.000,C 90.000,E1 61.769} C_DIS
LIN {X -0.298,Y -593.549,Z 1301.136,A 0.000,B 0.000,C 90.000,E1 60.461} C_DIS
LIN {X -0.289,Y -595.088,Z 1301.127,A 0.000,B 0.000,C 90.000,E1 58.869} C_DIS
LIN {X 0.186,Y -597.366,Z 1301.115,A 0.000,B 0.000,C 90.000,E1 56.707} C_DIS
LIN {X 0.073,Y -598.967,Z 1301.106,A 0.000,B 0.000,C 90.000,E1 55.135} C_DIS
LIN {X 0.081,Y -600.727,Z 1301.096,A 0.000,B 0.000,C 90.000,E1 53.290} C_DIS
LIN {X -0.228,Y -602.062,Z 1301.087,A 0.000,B 0.000,C 90.000,E1 51.743} C_DIS
LIN {X -0.288,Y -603.046,Z 1301.080,A 0.000,B 0.000,C 90.000,E1 50.436} C_DIS
LIN {X 0.045,Y -603.905,Z 1301.073,A 0.000,B 0.000,C 90.000,E1 49.094} C_DIS
LIN {X -0.316,Y -604.266,Z 1301.067,A 0.000,B 0.000,C 90.000,E1 48.081} C_DIS
LIN {X 0.234,Y -604.567,Z 1301.058,A 0.000,B 0.000,C 90.000,E1 46.458} C_DIS
LIN {X 0.107,Y -604.755,Z 1301.051,A 0.000,B 0.000,C 90.000,E1 45.162} C_DIS
LIN {X 0.181,Y -604.608,Z 1301.045,A 0.000,B 0.000,C 90.000,E1 44.109} C_DIS
LIN {X 0.046,Y -604.252,Z 1301.038,A 0.000,B 0.000,C 90.000,E1 42.813} C_DIS
LIN {X 0.137,Y -603.947,Z 1301.032,A 0.000,B 0.000,C 90.000,E1 41.757} C_DIS
LIN {X 0.230,Y -603.557,Z 1301.026,A 0.000,B 0.000,C 90.000,E1 40.701} C_DIS
LIN {X -0.021,Y -602.844,Z 1301.018,A 0.000,B 0.000,C 90.000,E1 39.152} C_DIS
LIN {X -0.199,Y -602.391,Z 1301.013,A 0.000,B 0.000,C 90.000,E1 38.382} C_DIS
LIN {X -0.262,Y -601.178,Z 1301.006,A 0.000,B 0.000,C 90.000,E1 37.076} C_DIS
LIN {X -0.113,Y -599.926,Z 1301.000,A 0.000,B 0.000,C 90.000,E1 36.011} C_DIS
LIN {X 0.019,Y -598.490,Z 1300.994,A 0.000,B 0.000,C 90.000,E1 34.945} C_DIS
LIN {X 0.012,Y -596.230,Z 1300.987,A 0.000,B 0.000,C 90.000,E1 33.627} C_DIS
LIN {X 0.247,Y -593.941,Z 1300.981,A 0.000,B 0.000,C 90.000,E1 32.546} C_DIS
LIN {X -0.254,Y -591.922,Z 1300.977,A 0.000,B 0.000,C 90.000,E1 31.799} C_DIS
LIN {X -0.271,Y -589.590,Z 1300.972,A 0.000,B 0.000,C 90.000,E1 31.003} C_DIS
LIN {X -0.193,Y -587.899,Z 1300.969,A 0.000,B 0.000,C 90.000,E1 30.463} C_DIS
LIN {X -0.251,Y -584.895,Z 1300.965,A 0.000,B 0.000,C 90.000,E1 29.667} C_DIS
LIN {X 0.297,Y -582.705,Z 1300.962,A 0.000,B 0.000,C 90.000,E1 29.077} C_DIS
LIN {X 0.111,Y -578.472,Z 1300.957,A 0.000,B 0.000,C 90.000,E1 28.153} C_DIS
LIN {X 0.184,Y -574.195,Z 1300.952,A 0.000,B 0.000,C 90.000,E1 27.334} C_DIS
LIN {X -0.034,Y -569.650,Z 1300.948,A 0.000,B 0.000,C 90.000,E1 26.539} C_DIS
LIN {X 0.042,Y -565.390,Z 1300.944,A 0.000,B 0.000,C 90.000,E1 25.848} C_DIS
LIN {X -0.114,Y -558.812,Z 1300.938,A 0.000,B 0.000,C 90.000,E1 24.899} C_DIS
LIN {X -0.128,Y -553.666,Z 1300.934,A 0.000,B 0.000,C 90.000,E1 24.207} C_DIS
LIN {X -0.189,Y -548.072,Z 1300.931,A 0.000,B 0.000,C 90.000,E1 23.515} C_DIS
LIN {X -0.048,Y -544.533,Z 1300.928,A 0.000,B 0.000,C 90.000,E1 23.078} C_DIS
LIN {X 0.031,Y -535.875,Z 1300.923,A 0.000,B 0.000,C 90.000,E1 22.078} C_DIS
LIN {X -0.183,Y -530.689,Z 1300.920,A 0.000,B 0.000,C 90.000,E1 21.535} C_DIS
LIN {X -0.191,Y -521.476,Z 1300.914,A 0.000,B 0.000,C 90.000,E1 20.556} C_DIS
LIN {X -0.143,Y -512.129,Z 1300.909,A 0.000,B 0.000,C 90.000,E1 19.577} C_DIS
LIN {X 0.144,Y -503.890,Z 1300.904,A 0.000,B 0.000,C 90.000,E1 18.725} C_DIS
LIN {X 0.004,Y -494.563,Z 1300.899,A 0.000,B 0.000,C 90.000,E1 17.819} C_DIS
LIN {X 0.185,Y -486.061,Z 1300.895,A 0.000,B 0.000,C 90.000,E1 16.985} C_DIS
LIN {X -0.014,Y -477.368,Z 1300.890,A 0.000,B 0.000,C 90.000,E1 16.205} C_DIS
LIN {X -0.116,Y -462.546,Z 1300.883,A 0.000,B 0.000,C 90.000,E1 14.883} C_DIS
LIN {X -0.193,Y -440.704,Z 1300.871,A 0.000,B 0.000,C 90.000,E1 12.827} C_DIS
LIN {X -0.057,Y -419.234,Z 1300.859,A 0.000,B 0.000,C 90.000,E1 10.602} C_DIS
LIN {X -0.146,Y -406.369,Z 1300.851,A 0.000,B 0.000,C 90.000,E1 9.208} C_DIS
LIN {X 0.096,Y -398.076,Z 1300.846,A 0.000,B 0.000,C 90.000,E1 8.219} C_DIS
LIN {X 0.118,Y -396.815,Z 1300.845,A 0.000,B 0.000,C 90.000,E1 8.049} C_DIS
LIN {X -0.174,Y -395.284,Z 1300.843,A 0.000,B 0.000,C 90.000,E1 7.814} C_DIS
LIN {X 0.180,Y -395.275,Z 1300.843,A 0.000,B 0.000,C 90.000,E1 7.757} C_DIS
LIN {X -0.101,Y -396.163,Z 1300.842,A 0.000,B 0.000,C 90.000,E1 7.644} C_DIS
LIN {X -0.079,Y -398.659,Z 1300.841,A 0.000,B 0.000,C 90.000,E1 7.409} C_DIS
LIN {X 0.111,Y -400.381,Z 1300.840,A 0.000,B 0.000,C 90.000,E1 7.239} C_DIS
LIN {X -0.032,Y -406.364,Z 1300.838,A 0.000,B 0.000,C 90.000,E1 6.891} C_DIS
LIN {X -0.169,Y -412.599,Z 1300.836,A 0.000,B 0.000,C 90.000,E1 6.543} C_DIS
LIN {X 0.037,Y -417.447,Z 1300.834,A 0.000,B 0.000,C 90.000,E1 6.201} C_DIS
LIN {X 0.081,Y -428.410,Z 1300.830,A 0.000,B 0.000,C 90.000,E1 5.391} C_DIS
LIN {X 0.234,Y -436.165,Z 1300.827,A 0.000,B 0.000,C 90.000,E1 4.759} C_DIS
LIN {X 0.129,Y -443.738,Z 1300.823,A 0.000,B 0.000,C 90.000,E1 4.131} C_DIS
LIN {X -0.216,Y -451.219,Z 1300.819,A 0.000,B 0.000,C 90.000,E1 3.498} C_DIS
LIN {X -0.062,Y -457.103,Z 1300.816,A 0.000,B 0.000,C 90.000,E1 2.922} C_DIS
LIN {X -0.220,Y -461.434,Z 1300.814,A 0.000,B 0.000,C 90.000,E1 2.522} C_DIS
LIN {X -0.113,Y -468.266,Z 1300.810,A 0.000,B 0.000,C 90.000,E1 1.776} C_DIS
LIN {X 0.114,Y -473.601,Z 1300.807,A 0.000,B 0.000,C 90.000,E1 1.146} C_DIS
LIN {X 0.111,Y -480.845,Z 1300.801,A 0.000,B 0.000,C 90.000,E1 0.229} C_DIS
LIN {X 0.156,Y -487.363,Z 1300.796,A 0.000,B 0.000,C 90.000,E1 359.312} C_DIS
LIN {X -0.181,Y -491.469,Z 1300.793,A 0.000,B 0.000,C 90.000,E1 358.740} C_DIS
LIN {X -0.128,Y -497.054,Z 1300.788,A 0.000,B 0.000,C 90.000,E1 357.822} C_DIS
LIN {X -0.031,Y -502.177,Z 1300.783,A 0.000,B 0.000,C 90.000,E1 356.906} C_DIS
LIN {X -0.243,Y -505.391,Z 1300.780,A 0.000,B 0.000,C 90.000,E1 356.331} C_DIS
LIN {X -0.028,Y -509.930,Z 1300.775,A 0.000,B 0.000,C 90.000,E1 355.412} C_DIS
LIN {X -0.226,Y -514.111,Z 1300.770,A 0.000,B 0.000,C 90.000,E1 354.546} C_DIS
LIN {X 0.085,Y -517.912,Z 1300.765,A 0.000,B 0.000,C 90.000,E1 353.628} C_DIS
LIN {X -0.231,Y -519.769,Z 1300.762,A 0.000,B 0.000,C 90.000,E1 353.223} C_DIS
LIN {X 0.196,Y -523.068,Z 1300.757,A 0.000,B 0.000,C 90.000,E1 352.299} C_DIS
LIN {X 0.130,Y -525.166,Z 1300.754,A 0.000,B 0.000,C 90.000,E1 351.724} C_DIS
LIN {X 0.175,Y -528.023,Z 1300.749,A 0.000,B 0.000,C 90.000,E1 350.849} C_DIS
LIN {X 0.170,Y -530.645,Z 1300.745,A 0.000,B 0.000,C 90.000,E1 349.982} C_DIS
LIN {X -0.196,Y -533.717,Z 1300.738,A 0.000,B 0.000,C 90.000,E1 348.870} C_DIS
LIN {X -0.046,Y -535.831,Z 1300.733,A 0.000,B 0.000,C 90.000,E1 347.993} C_DIS
LIN {X 0.125,Y -537.624,Z 1300.729,A 0.000,B 0.000,C 90.000,E1 347.117} C_DIS
LIN {X -0.020,Y -539.708,Z 1300.722,A 0.000,B 0.000,C 90.000,E1 345.992} C_DIS
LIN {X 0.182,Y -541.019,Z 1300.718,A 0.000,B 0.000,C 90.000,E1 345.117} C_DIS
LIN {X 0.010,Y -542.057,Z 1300.713,A 0.000,B 0.000,C 90.000,E1 344.283} C_DIS
LIN {X 0.075,Y -543.109,Z 1300.706,A 0.000,B 0.000,C 90.000,E1 343.142} C_DIS
LIN {X -0.074,Y -543.608,Z 1300.702,A 0.000,B 0.000,C 90.000,E1 342.308} C_DIS
LIN {X -0.053,Y -543.841,Z 1300.697,A 0.000,B 0.000,C 90.000,E1 341.456} C_DIS
LIN {X -0.265,Y -543.827,Z 1300.694,A 0.000,B 0.000,C 90.000,E1 340.913} C_DIS
LIN {X -0.237,Y -543.509,Z 1300.689,A 0.000,B 0.000,C 90.000,E1 340.061} C_DIS
LIN {X -0.213,Y -542.982,Z 1300.684,A 0.000,B 0.000,C 90.000,E1 339.209} C_DIS
LIN {X 0.265,Y -542.455,Z 1300.681,A 0.000,B 0.000,C 90.000,E1 338.592} C_DIS
LIN {X -0.036,Y -540.020,Z 1300.672,A 0.000,B 0.000,C 90.000,E1 336.922} C_DIS
LIN {X 0.192,Y -539.469,Z 1300.670,A 0.000,B 0.000,C 90.000,E1 336.613} C_DIS
LIN {X -0.125,Y -537.512,Z 1300.666,A 0.000,B 0.000,C 90.000,E1 335.793} C_DIS
LIN {X 0.180,Y -533.571,Z 1300.658,A 0.000,B 0.000,C 90.000,E1 334.332} C_DIS
LIN {X -0.192,Y -527.029,Z 1300.646,A 0.000,B 0.000,C 90.000,E1 332.359} C_DIS
LIN {X 0.062,Y -523.961,Z 1300.642,A 0.000,B 0.000,C 90.000,E1 331.463} C_DIS
LIN {X -0.248,Y -519.397,Z 1300.635,A 0.000,B 0.000,C 90.000,E1 330.333} C_DIS
LIN {X 0.164,Y -515.525,Z 1300.630,A 0.000,B 0.000,C 90.000,E1 329.410} C_DIS
LIN {X -0.187,Y -509.311,Z 1300.623,A 0.000,B 0.000,C 90.000,E1 328.122} C_DIS
LIN {X -0.015,Y -503.696,Z 1300.616,A 0.000,B 0.000,C 90.000,E1 326.914} C_DIS
LIN {X -0.322,Y -501.746,Z 1300.614,A 0.000,B 0.000,C 90.000,E1 326.501} C_DIS
LIN {X -0.144,Y -499.598,Z 1300.610,A 0.000,B 0.000,C 90.000,E1 325.881} C_DIS
LIN {X -0.267,Y -498.691,Z 1300.609,A 0.000,B 0.000,C 90.000,E1 325.595} C_DIS
LIN {X -0.143,Y -496.583,Z 1300.604,A 0.000,B 0.000,C 90.000,E1 324.689} C_DIS
LIN {X -0.146,Y -495.134,Z 1300.599,A 0.000,B 0.000,C 90.000,E1 323.783} C_DIS
LIN {X -0.159,Y -493.798,Z 1300.590,A 0.000,B 0.000,C 90.000,E1 322.271} C_DIS
LIN {X -0.051,Y -493.299,Z 1300.584,A 0.000,B 0.000,C 90.000,E1 321.045} C_DIS
LIN {X -0.137,Y -493.405,Z 1300.568,A 0.000,B 0.000,C 90.000,E1 318.324} C_DIS
LIN {X 0.055,Y -493.447,Z 1300.563,A 0.000,B 0.000,C 90.000,E1 317.391} C_DIS
LIN {X 0.247,Y -493.075,Z 1300.558,A 0.000,B 0.000,C 90.000,E1 316.458} C_DIS
LIN {X -0.097,Y -492.542,Z 1300.555,A 0.000,B 0.000,C 90.000,E1 315.891} C_DIS
LIN {X 0.253,Y -491.677,Z 1300.552,A 0.000,B 0.000,C 90.000,E1 315.243} C_DIS
LIN {X -0.269,Y -491.028,Z 1300.550,A 0.000,B 0.000,C 90.000,E1 315.000} C_DIS
LIN {X -0.098,Y -490.162,Z 1300.548,A 0.000,B 0.000,C 90.000,E1 314.676} C_DIS
LIN {X -0.013,Y -489.587,Z 1300.547,A 0.000,B 0.000,C 90.000,E1 314.514} C_DIS
LIN {X 0.071,Y -488.828,Z 1300.547,A 0.000,B 0.000,C 90.000,E1 314.352} C_DIS
LIN {X 0.308,Y -485.126,Z 1300.544,A 0.000,B 0.000,C 90.000,E1 313.866} C_DIS
LIN {X -0.124,Y -465.813,Z 1300.530,A 0.000,B 0.000,C 90.000,E1 311.434} C_DIS
LIN {X 0.277,Y -448.335,Z 1300.516,A 0.000,B 0.000,C 90.000,E1 308.830} C_DIS
LIN {X -0.040,Y -432.573,Z 1300.501,A 0.000,B 0.000,C 90.000,E1 306.251} C_DIS
LIN {X -0.117,Y -418.419,Z 1300.486,A 0.000,B 0.000,C 90.000,E1 303.579} C_DIS
LIN {X 0.171,Y -405.774,Z 1300.471,A 0.000,B 0.000,C 90.000,E1 300.797} C_DIS
LIN {X 0.176,Y -396.890,Z 1300.459,A 0.000,B 0.000,C 90.000,E1 298.615} C_DIS
LIN {X 0.139,Y -396.886,Z 1300.459,A 0.000,B 0.000,C 90.000,E1 298.615} C_DIS
LIN {X -0.116,Y -397.532,Z 1300.453,A 0.000,B 0.000,C 90.000,E1 297.513} C_DIS
LIN {X -0.130,Y -401.353,Z 1300.427,A 0.000,B 0.000,C 90.000,E1 292.950} C_DIS
LIN {X -0.050,Y -401.658,Z 1300.426,A 0.000,B 0.000,C 90.000,E1 292.589} C_DIS
LIN {X 0.102,Y -404.749,Z 1300.395,A 0.000,B 0.000,C 90.000,E1 286.985} C_DIS
LIN {X 0.115,Y -406.156,Z 1300.364,A 0.000,B 0.000,C 90.000,E1 281.422} C_DIS
LIN {X -0.184,Y -405.675,Z 1300.333,A 0.000,B 0.000,C 90.000,E1 275.910} C_DIS
LIN {X -0.112,Y -403.564,Z 1300.306,A 0.000,B 0.000,C 90.000,E1 271.031} C_DIS
LIN {X -0.177,Y -403.170,Z 1300.302,A 0.000,B 0.000,C 90.000,E1 270.344} C_DIS
LIN {X 0.057,Y -399.062,Z 1300.273,A 0.000,B 0.000,C 90.000,E1 265.065} C_DIS
LIN {X -0.003,Y -398.763,Z 1300.271,A 0.000,B 0.000,C 90.000,E1 264.723} C_DIS
LIN {X -0.112,Y -393.284,Z 1300.243,A 0.000,B 0.000,C 90.000,E1 259.803} C_DIS
LIN {X -0.191,Y -392.656,Z 1300.239,A 0.000,B 0.000,C 90.000,E1 259.106} C_DIS
LIN {X -0.020,Y -386.237,Z 1300.214,A 0.000,B 0.000,C 90.000,E1 254.448} C_DIS
LIN {X -0.054,Y -385.139,Z 1300.208,A 0.000,B 0.000,C 90.000,E1 253.378} C_DIS
LIN {X 0.054,Y -377.803,Z 1300.182,A 0.000,B 0.000,C 90.000,E1 248.666} C_DIS
LIN {X 0.034,Y -376.740,Z 1300.177,A 0.000,B 0.000,C 90.000,E1 247.794} C_DIS
LIN {X -0.004,Y -376.736,Z 1300.177,A 0.000,B 0.000,C 90.000,E1 247.794} C_DIS
LIN {X 0.130,Y -386.141,Z 1300.159,A 0.000,B 0.000,C 90.000,E1 244.665} C_DIS
LIN {X 0.101,Y -396.928,Z 1300.143,A 0.000,B 0.000,C 90.000,E1 241.641} C_DIS
LIN {X 0.155,Y -409.261,Z 1300.126,A 0.000,B 0.000,C 90.000,E1 238.663} C_DIS
LIN {X 0.121,Y -422.373,Z 1300.111,A 0.000,B 0.000,C 90.000,E1 235.928} C_DIS
LIN {X 0.065,Y -437.034,Z 1300.096,A 0.000,B 0.000,C 90.000,E1 233.256} C_DIS
LIN {X 0.063,Y -450.102,Z 1300.084,A 0.000,B 0.000,C 90.000,E1 231.126} C_DIS
LIN {X 0.054,Y -450.786,Z 1300.083,A 0.000,B 0.000,C 90.000,E1 230.964} C_DIS
LIN {X 0.045,Y -451.690,Z 1300.081,A 0.000,B 0.000,C 90.000,E1 230.642} C_DIS
LIN {X -0.246,Y -452.306,Z 1300.080,A 0.000,B 0.000,C 90.000,E1 230.356} C_DIS
LIN {X 0.101,Y -452.761,Z 1300.078,A 0.000,B 0.000,C 90.000,E1 229.989} C_DIS
LIN {X -0.182,Y -453.328,Z 1300.074,A 0.000,B 0.000,C 90.000,E1 229.380} C_DIS
LIN {X -0.106,Y -453.702,Z 1300.069,A 0.000,B 0.000,C 90.000,E1 228.405} C_DIS
LIN {X 0.277,Y -453.621,Z 1300.063,A 0.000,B 0.000,C 90.000,E1 227.391} C_DIS
LIN {X 0.050,Y -453.358,Z 1300.055,A 0.000,B 0.000,C 90.000,E1 225.810} C_DIS
LIN {X 0.168,Y -453.195,Z 1300.042,A 0.000,B 0.000,C 90.000,E1 223.542} C_DIS
LIN {X -0.310,Y -455.225,Z 1300.010,A 0.000,B 0.000,C 90.000,E1 217.810} C_DIS
LIN {X -0.037,Y -456.368,Z 1300.001,A 0.000,B 0.000,C 90.000,E1 216.171} C_DIS
LIN {X 0.208,Y -458.532,Z 1299.987,A 0.000,B 0.000,C 90.000,E1 213.579} C_DIS
LIN {X 0.022,Y -461.945,Z 1299.969,A 0.000,B 0.000,C 90.000,E1 210.413} C_DIS
LIN {X 0.058,Y -463.979,Z 1299.960,A 0.000,B 0.000,C 90.000,E1 208.821} C_DIS
LIN {X 0.114,Y -467.350,Z 1299.946,A 0.000,B 0.000,C 90.000,E1 206.283} C_DIS
LIN {X 0.171,Y -470.092,Z 1299.936,A 0.000,B 0.000,C 90.000,E1 204.387} C_DIS
LIN {X 0.137,Y -472.374,Z 1299.927,A 0.000,B 0.000,C 90.000,E1 202.823} C_DIS
LIN {X -0.122,Y -476.000,Z 1299.913,A 0.000,B 0.000,C 90.000,E1 200.355} C_DIS
LIN {X 0.052,Y -478.459,Z 1299.904,A 0.000,B 0.000,C 90.000,E1 198.779} C_DIS
LIN {X 0.113,Y -481.380,Z 1299.894,A 0.000,B 0.000,C 90.000,E1 196.913} C_DIS
LIN {X 0.112,Y -483.817,Z 1299.885,A 0.000,B 0.000,C 90.000,E1 195.371} C_DIS
LIN {X 0.160,Y -486.231,Z 1299.877,A 0.000,B 0.000,C 90.000,E1 193.828} C_DIS
LIN {X 0.254,Y -488.166,Z 1299.870,A 0.000,B 0.000,C 90.000,E1 192.591} C_DIS
LIN {X 0.057,Y -491.033,Z 1299.860,A 0.000,B 0.000,C 90.000,E1 190.782} C_DIS
LIN {X -0.080,Y -493.838,Z 1299.850,A 0.000,B 0.000,C 90.000,E1 188.973} C_DIS
LIN {X -0.154,Y -496.170,Z 1299.841,A 0.000,B 0.000,C 90.000,E1 187.466} C_DIS
LIN {X 0.243,Y -498.483,Z 1299.833,A 0.000,B 0.000,C 90.000,E1 185.910} C_DIS
LIN {X -0.222,Y -500.267,Z 1299.826,A 0.000,B 0.000,C 90.000,E1 184.759} C_DIS
LIN {X 0.084,Y -502.718,Z 1299.816,A 0.000,B 0.000,C 90.000,E1 182.922} C_DIS
LIN {X 0.240,Y -503.899,Z 1299.811,A 0.000,B 0.000,C 90.000,E1 182.007} C_DIS
LIN {X 0.213,Y -505.557,Z 1299.803,A 0.000,B 0.000,C 90.000,E1 180.516} C_DIS
LIN {X 0.206,Y -507.110,Z 1299.795,A 0.000,B 0.000,C 90.000,E1 179.026} C_DIS
LIN {X -0.077,Y -507.840,Z 1299.790,A 0.000,B 0.000,C 90.000,E1 178.165} C_DIS
LIN {X -0.029,Y -508.858,Z 1299.781,A 0.000,B 0.000,C 90.000,E1 176.674} C_DIS
LIN {X 0.124,Y -509.441,Z 1299.775,A 0.000,B 0.000,C 90.000,E1 175.469} C_DIS
LIN {X -0.186,Y -509.725,Z 1299.768,A 0.000,B 0.000,C 90.000,E1 174.318} C_DIS
LIN {X -0.032,Y -509.678,Z 1299.760,A 0.000,B 0.000,C 90.000,E1 172.818} C_DIS
LIN {X -0.187,Y -509.575,Z 1299.757,A 0.000,B 0.000,C 90.000,E1 172.243} C_DIS
LIN {X 0.113,Y -509.106,Z 1299.752,A 0.000,B 0.000,C 90.000,E1 171.319} C_DIS
LIN {X -0.016,Y -508.383,Z 1299.747,A 0.000,B 0.000,C 90.000,E1 170.443} C_DIS
LIN {X -0.103,Y -507.908,Z 1299.744,A 0.000,B 0.000,C 90.000,E1 169.859} C_DIS
LIN {X 0.216,Y -506.501,Z 1299.737,A 0.000,B 0.000,C 90.000,E1 168.634} C_DIS
LIN {X 0.014,Y -504.570,Z 1299.730,A 0.000,B 0.000,C 90.000,E1 167.465} C_DIS
LIN {X -0.105,Y -502.215,Z 1299.724,A 0.000,B 0.000,C 90.000,E1 166.284} C_DIS
LIN {X -0.238,Y -500.900,Z 1299.720,A 0.000,B 0.000,C 90.000,E1 165.700} C_DIS
LIN {X 0.112,Y -497.245,Z 1299.712,A 0.000,B 0.000,C 90.000,E1 164.157} C_DIS
LIN {X 0.014,Y -494.294,Z 1299.705,A 0.000,B 0.000,C 90.000,E1 162.960} C_DIS
LIN {X -0.051,Y -492.622,Z 1299.702,A 0.000,B 0.000,C 90.000,E1 162.362} C_DIS
LIN {X -0.129,Y -490.674,Z 1299.699,A 0.000,B 0.000,C 90.000,E1 161.764} C_DIS
LIN {X -0.176,Y -486.481,Z 1299.692,A 0.000,B 0.000,C 90.000,E1 160.550} C_DIS
LIN {X -0.126,Y -483.080,Z 1299.687,A 0.000,B 0.000,C 90.000,E1 159.625} C_DIS
LIN {X -0.282,Y -480.178,Z 1299.682,A 0.000,B 0.000,C 90.000,E1 158.720} C_DIS
LIN {X -0.284,Y -479.405,Z 1299.680,A 0.000,B 0.000,C 90.000,E1 158.411} C_DIS
LIN {X 0.153,Y -478.870,Z 1299.678,A 0.000,B 0.000,C 90.000,E1 158.050} C_DIS
LIN {X -0.086,Y -478.512,Z 1299.676,A 0.000,B 0.000,C 90.000,E1 157.614} C_DIS
LIN {X 0.085,Y -479.521,Z 1299.672,A 0.000,B 0.000,C 90.000,E1 156.922} C_DIS
LIN {X 0.073,Y -480.350,Z 1299.670,A 0.000,B 0.000,C 90.000,E1 156.613} C_DIS
LIN {X -0.017,Y -481.458,Z 1299.669,A 0.000,B 0.000,C 90.000,E1 156.433} C_DIS
LIN {X -0.154,Y -484.038,Z 1299.667,A 0.000,B 0.000,C 90.000,E1 156.102} C_DIS
LIN {X -0.261,Y -486.183,Z 1299.666,A 0.000,B 0.000,C 90.000,E1 155.921} C_DIS
LIN {X 0.124,Y -488.691,Z 1299.665,A 0.000,B 0.000,C 90.000,E1 155.613} C_DIS
LIN {X 0.168,Y -497.568,Z 1299.660,A 0.000,B 0.000,C 90.000,E1 154.793} C_DIS
LIN {X -0.168,Y -504.441,Z 1299.656,A 0.000,B 0.000,C 90.000,E1 154.152} C_DIS
LIN {X -0.108,Y -510.951,Z 1299.652,A 0.000,B 0.000,C 90.000,E1 153.435} C_DIS
LIN {X -0.176,Y -514.785,Z 1299.650,A 0.000,B 0.000,C 90.000,E1 152.999} C_DIS
LIN {X -0.062,Y -519.358,Z 1299.647,A 0.000,B 0.000,C 90.000,E1 152.410} C_DIS
LIN {X -0.004,Y -523.507,Z 1299.643,A 0.000,B 0.000,C 90.000,E1 151.820} C_DIS
LIN {X -0.167,Y -527.220,Z 1299.640,A 0.000,B 0.000,C 90.000,E1 151.257} C_DIS
LIN {X -0.066,Y -530.354,Z 1299.637,A 0.000,B 0.000,C 90.000,E1 150.667} C_DIS
LIN {X -0.091,Y -533.534,Z 1299.633,A 0.000,B 0.000,C 90.000,E1 149.950} C_DIS
LIN {X 0.325,Y -535.636,Z 1299.630,A 0.000,B 0.000,C 90.000,E1 149.331} C_DIS
LIN {X 0.025,Y -537.459,Z 1299.627,A 0.000,B 0.000,C 90.000,E1 148.791} C_DIS
LIN {X 0.198,Y -538.965,Z 1299.624,A 0.000,B 0.000,C 90.000,E1 148.201} C_DIS
LIN {X 0.201,Y -539.878,Z 1299.622,A 0.000,B 0.000,C 90.000,E1 147.916} C_DIS
LIN {X -0.079,Y -540.516,Z 1299.620,A 0.000,B 0.000,C 90.000,E1 147.661} C_DIS
LIN {X -0.004,Y -540.775,Z 1299.620,A 0.000,B 0.000,C 90.000,E1 147.582} C_DIS
LIN {X 0.071,Y -541.278,Z 1299.620,A 0.000,B 0.000,C 90.000,E1 147.502} C_DIS
LIN {X -0.068,Y -542.774,Z 1299.619,A 0.000,B 0.000,C 90.000,E1 147.375} C_DIS
LIN {X -0.106,Y -546.113,Z 1299.617,A 0.000,B 0.000,C 90.000,E1 147.120} C_DIS
LIN {X 0.133,Y -560.024,Z 1299.613,A 0.000,B 0.000,C 90.000,E1 146.342} C_DIS
LIN {X 0.118,Y -562.979,Z 1299.612,A 0.000,B 0.000,C 90.000,E1 146.167} C_DIS
LIN {X -0.175,Y -571.816,Z 1299.609,A 0.000,B 0.000,C 90.000,E1 145.595} C_DIS
LIN {X -0.093,Y -579.192,Z 1299.606,A 0.000,B 0.000,C 90.000,E1 145.055} C_DIS
LIN {X -0.008,Y -584.889,Z 1299.603,A 0.000,B 0.000,C 90.000,E1 144.609} C_DIS
LIN {X 0.089,Y -590.250,Z 1299.601,A 0.000,B 0.000,C 90.000,E1 144.149} C_DIS
LIN {X 0.097,Y -597.929,Z 1299.597,A 0.000,B 0.000,C 90.000,E1 143.417} C_DIS
LIN {X -0.127,Y -602.711,Z 1299.594,A 0.000,B 0.000,C 90.000,E1 142.924} C_DIS
LIN {X -0.089,Y -607.143,Z 1299.591,A 0.000,B 0.000,C 90.000,E1 142.396} C_DIS
LIN {X -0.400,Y -611.235,Z 1299.588,A 0.000,B 0.000,C 90.000,E1 141.904} C_DIS
LIN {X 0.173,Y -614.952,Z 1299.585,A 0.000,B 0.000,C 90.000,E1 141.331} C_DIS
LIN {X -0.227,Y -619.266,Z 1299.582,A 0.000,B 0.000,C 90.000,E1 140.723} C_DIS
LIN {X -0.111,Y -623.301,Z 1299.578,A 0.000,B 0.000,C 90.000,E1 140.070} C_DIS
LIN {X 0.070,Y -626.400,Z 1299.575,A 0.000,B 0.000,C 90.000,E1 139.542} C_DIS
LIN {X 0.024,Y -631.779,Z 1299.570,A 0.000,B 0.000,C 90.000,E1 138.528} C_DIS
LIN {X 0.128,Y -636.122,Z 1299.565,A 0.000,B 0.000,C 90.000,E1 137.634} C_DIS
LIN {X 0.211,Y -640.849,Z 1299.559,A 0.000,B 0.000,C 90.000,E1 136.620} C_DIS
LIN {X -0.184,Y -646.565,Z 1299.552,A 0.000,B 0.000,C 90.000,E1 135.405} C_DIS
LIN {X 0.435,Y -652.003,Z 1299.545,A 0.000,B 0.000,C 90.000,E1 134.109} C_DIS
LIN {X -0.234,Y -657.318,Z 1299.538,A 0.000,B 0.000,C 90.000,E1 132.933} C_DIS
LIN {X 0.110,Y -662.536,Z 1299.532,A 0.000,B 0.000,C 90.000,E1 131.676} C_DIS
LIN {X 0.117,Y -665.511,Z 1299.528,A 0.000,B 0.000,C 90.000,E1 130.943} C_DIS
LIN {X -0.355,Y -669.317,Z 1299.522,A 0.000,B 0.000,C 90.000,E1 130.011} C_DIS
LIN {X 0.247,Y -672.844,Z 1299.517,A 0.000,B 0.000,C 90.000,E1 128.991} C_DIS
LIN {X -0.033,Y -677.044,Z 1299.510,A 0.000,B 0.000,C 90.000,E1 127.810} C_DIS
LIN {X -0.275,Y -680.076,Z 1299.505,A 0.000,B 0.000,C 90.000,E1 126.870} C_DIS
LIN {X 0.082,Y -683.489,Z 1299.498,A 0.000,B 0.000,C 90.000,E1 125.644} C_DIS
LIN {X 0.076,Y -685.995,Z 1299.493,A 0.000,B 0.000,C 90.000,E1 124.692} C_DIS
LIN {X -0.458,Y -688.251,Z 1299.488,A 0.000,B 0.000,C 90.000,E1 123.785} C_DIS
LIN {X -0.018,Y -690.218,Z 1299.482,A 0.000,B 0.000,C 90.000,E1 122.801} C_DIS
LIN {X 0.293,Y -692.274,Z 1299.476,A 0.000,B 0.000,C 90.000,E1 121.592} C_DIS
LIN {X -0.068,Y -694.442,Z 1299.468,A 0.000,B 0.000,C 90.000,E1 120.207} C_DIS
LIN {X 0.073,Y -695.458,Z 1299.464,A 0.000,B 0.000,C 90.000,E1 119.489} C_DIS
LIN {X -0.384,Y -696.280,Z 1299.460,A 0.000,B 0.000,C 90.000,E1 118.821} C_DIS
LIN {X -0.226,Y -696.973,Z 1299.456,A 0.000,B 0.000,C 90.000,E1 118.103} C_DIS
LIN {X -0.063,Y -697.450,Z 1299.452,A 0.000,B 0.000,C 90.000,E1 117.385} C_DIS
LIN {X 0.101,Y -697.679,Z 1299.448,A 0.000,B 0.000,C 90.000,E1 116.668} C_DIS
LIN {X -0.046,Y -697.704,Z 1299.444,A 0.000,B 0.000,C 90.000,E1 115.976} C_DIS
LIN {X -0.189,Y -697.314,Z 1299.440,A 0.000,B 0.000,C 90.000,E1 115.283} C_DIS
LIN {X 0.334,Y -696.863,Z 1299.438,A 0.000,B 0.000,C 90.000,E1 114.771} C_DIS
LIN {X -0.071,Y -696.049,Z 1299.435,A 0.000,B 0.000,C 90.000,E1 114.335} C_DIS
LIN {X 0.437,Y -694.564,Z 1299.433,A 0.000,B 0.000,C 90.000,E1 113.823} C_DIS
LIN {X -0.227,Y -693.659,Z 1299.431,A 0.000,B 0.000,C 90.000,E1 113.643} C_DIS
LIN {X -0.012,Y -690.551,Z 1299.429,A 0.000,B 0.000,C 90.000,E1 113.153} C_DIS
LIN {X 0.106,Y -689.657,Z 1299.428,A 0.000,B 0.000,C 90.000,E1 113.025} C_DIS
LIN {X 0.222,Y -688.318,Z 1299.427,A 0.000,B 0.000,C 90.000,E1 112.898} C_DIS
LIN {X 0.070,Y -682.429,Z 1299.425,A 0.000,B 0.000,C 90.000,E1 112.514} C_DIS
LIN {X 0.165,Y -680.434,Z 1299.425,A 0.000,B 0.000,C 90.000,E1 112.408} C_DIS
LIN {X -0.132,Y -675.635,Z 1299.424,A 0.000,B 0.000,C 90.000,E1 112.280} C_DIS
LIN {X 0.154,Y -671.767,Z 1299.423,A 0.000,B 0.000,C 90.000,E1 112.153} C_DIS
LIN {X -0.129,Y -664.034,Z 1299.423,A 0.000,B 0.000,C 90.000,E1 112.078} C_DIS
LIN {X 0.103,Y -656.546,Z 1299.422,A 0.000,B 0.000,C 90.000,E1 112.025} C_DIS
LIN {X 0.041,Y -653.442,Z 1299.422,A 0.000,B 0.000,C 90.000,E1 112.025} C_DIS
LIN {X -0.022,Y -649.209,Z 1299.422,A 0.000,B 0.000,C 90.000,E1 112.025} C_DIS
LIN {X 0.022,Y -644.369,Z 1299.422,A 0.000,B 0.000,C 90.000,E1 111.972} C_DIS
LIN {X -0.193,Y -642.518,Z 1299.422,A 0.000,B 0.000,C 90.000,E1 111.950} C_DIS
LIN {X -0.303,Y -640.463,Z 1299.422,A 0.000,B 0.000,C 90.000,E1 111.897} C_DIS
LIN {X 0.254,Y -640.478,Z 1299.422,A 0.000,B 0.000,C 90.000,E1 111.844} C_DIS
LIN {X -0.141,Y -642.204,Z 1299.420,A 0.000,B 0.000,C 90.000,E1 111.535} C_DIS
LIN {X 0.147,Y -650.547,Z 1299.414,A 0.000,B 0.000,C 90.000,E1 110.429} C_DIS
LIN {X -0.051,Y -655.430,Z 1299.410,A 0.000,B 0.000,C 90.000,E1 109.704} C_DIS
LIN {X -0.035,Y -658.929,Z 1299.406,A 0.000,B 0.000,C 90.000,E1 109.087} C_DIS
LIN {X -0.047,Y -661.463,Z 1299.403,A 0.000,B 0.000,C 90.000,E1 108.598} C_DIS
LIN {X -0.255,Y -663.757,Z 1299.401,A 0.000,B 0.000,C 90.000,E1 108.127} C_DIS
LIN {X -0.333,Y -666.813,Z 1299.397,A 0.000,B 0.000,C 90.000,E1 107.402} C_DIS
LIN {X 0.258,Y -669.391,Z 1299.393,A 0.000,B 0.000,C 90.000,E1 106.622} C_DIS
LIN {X 0.113,Y -670.927,Z 1299.390,A 0.000,B 0.000,C 90.000,E1 106.150} C_DIS
LIN {X 0.036,Y -673.380,Z 1299.384,A 0.000,B 0.000,C 90.000,E1 105.190} C_DIS
LIN {X -0.081,Y -674.435,Z 1299.382,A 0.000,B 0.000,C 90.000,E1 104.717} C_DIS
LIN {X -0.293,Y -676.145,Z 1299.376,A 0.000,B 0.000,C 90.000,E1 103.772} C_DIS
LIN {X 0.220,Y -676.915,Z 1299.372,A 0.000,B 0.000,C 90.000,E1 103.008} C_DIS
LIN {X 0.080,Y -677.389,Z 1299.368,A 0.000,B 0.000,C 90.000,E1 102.299} C_DIS
LIN {X 0.033,Y -677.522,Z 1299.367,A 0.000,B 0.000,C 90.000,E1 102.063} C_DIS
LIN {X -0.244,Y -677.414,Z 1299.363,A 0.000,B 0.000,C 90.000,E1 101.366} C_DIS
LIN {X -0.339,Y -677.148,Z 1299.360,A 0.000,B 0.000,C 90.000,E1 100.894} C_DIS
LIN {X 0.224,Y -676.701,Z 1299.358,A 0.000,B 0.000,C 90.000,E1 100.366} C_DIS
LIN {X -0.058,Y -675.492,Z 1299.354,A 0.000,B 0.000,C 90.000,E1 99.670} C_DIS
LIN {X -0.287,Y -674.437,Z 1299.351,A 0.000,B 0.000,C 90.000,E1 99.208} C_DIS
LIN {X 0.148,Y -673.043,Z 1299.348,A 0.000,B 0.000,C 90.000,E1 98.690} C_DIS
LIN {X 0.008,Y -671.251,Z 1299.346,A 0.000,B 0.000,C 90.000,E1 98.219} C_DIS
LIN {X 0.247,Y -667.931,Z 1299.342,A 0.000,B 0.000,C 90.000,E1 97.473} C_DIS
LIN {X 0.063,Y -665.503,Z 1299.339,A 0.000,B 0.000,C 90.000,E1 97.004} C_DIS
LIN {X 0.149,Y -660.547,Z 1299.334,A 0.000,B 0.000,C 90.000,E1 96.144} C_DIS
LIN {X -0.265,Y -656.597,Z 1299.331,A 0.000,B 0.000,C 90.000,E1 95.568} C_DIS
LIN {X -0.057,Y -652.054,Z 1299.327,A 0.000,B 0.000,C 90.000,E1 94.935} C_DIS
LIN {X 0.219,Y -648.107,Z 1299.325,A 0.000,B 0.000,C 90.000,E1 94.416} C_DIS
LIN {X 0.112,Y -640.262,Z 1299.320,A 0.000,B 0.000,C 90.000,E1 93.555} C_DIS
LIN {X 0.298,Y -635.544,Z 1299.317,A 0.000,B 0.000,C 90.000,E1 93.037} C_DIS
LIN {X 0.088,Y -627.085,Z 1299.312,A 0.000,B 0.000,C 90.000,E1 92.178} C_DIS
LIN {X -0.236,Y -621.977,Z 1299.309,A 0.000,B 0.000,C 90.000,E1 91.718} C_DIS
LIN {X -0.300,Y -616.456,Z 1299.307,A 0.000,B 0.000,C 90.000,E1 91.260} C_DIS
LIN {X 0.054,Y -609.006,Z 1299.304,A 0.000,B 0.000,C 90.000,E1 90.688} C_DIS
LIN {X 0.058,Y -602.626,Z 1299.302,A 0.000,B 0.000,C 90.000,E1 90.286} C_DIS
LIN {X -0.206,Y -595.873,Z 1299.300,A 0.000,B 0.000,C 90.000,E1 89.943} C_DIS
LIN {X -0.043,Y -588.824,Z 1299.298,A 0.000,B 0.000,C 90.000,E1 89.599} C_DIS
LIN {X -0.081,Y -577.766,Z 1299.296,A 0.000,B 0.000,C 90.000,E1 89.198} C_DIS
LIN {X -0.138,Y -572.274,Z 1299.294,A 0.000,B 0.000,C 90.000,E1 88.969} C_DIS
LIN {X 0.160,Y -570.932,Z 1299.294,A 0.000,B 0.000,C 90.000,E1 88.854} C_DIS
LIN {X 0.113,Y -570.882,Z 1299.294,A 0.000,B 0.000,C 90.000,E1 88.854} C_DIS
LIN {X -0.143,Y -569.980,Z 1299.293,A 0.000,B 0.000,C 90.000,E1 88.682} C_DIS
LIN {X -0.234,Y -569.833,Z 1299.290,A 0.000,B 0.000,C 90.000,E1 88.282} C_DIS
LIN {X -0.131,Y -571.802,Z 1299.277,A 0.000,B 0.000,C 90.000,E1 85.812} C_DIS
LIN {X -0.089,Y -574.151,Z 1299.265,A 0.000,B 0.000,C 90.000,E1 83.628} C_DIS
LIN {X 0.178,Y -575.747,Z 1299.257,A 0.000,B 0.000,C 90.000,E1 82.243} C_DIS
LIN {X -0.034,Y -578.360,Z 1299.245,A 0.000,B 0.000,C 90.000,E1 80.095} C_DIS
LIN {X 0.169,Y -579.561,Z 1299.239,A 0.000,B 0.000,C 90.000,E1 78.993} C_DIS
LIN {X 0.153,Y -580.836,Z 1299.231,A 0.000,B 0.000,C 90.000,E1 77.645} C_DIS
LIN {X -0.070,Y -581.840,Z 1299.225,A 0.000,B 0.000,C 90.000,E1 76.589} C_DIS
LIN {X 0.090,Y -582.861,Z 1299.218,A 0.000,B 0.000,C 90.000,E1 75.227} C_DIS
LIN {X -0.294,Y -583.816,Z 1299.211,A 0.000,B 0.000,C 90.000,E1 73.921} C_DIS
LIN {X -0.272,Y -584.873,Z 1299.202,A 0.000,B 0.000,C 90.000,E1 72.308} C_DIS
LIN {X -0.053,Y -585.958,Z 1299.193,A 0.000,B 0.000,C 90.000,E1 70.678} C_DIS
LIN {X 0.255,Y -587.081,Z 1299.182,A 0.000,B 0.000,C 90.000,E1 68.773} C_DIS
LIN {X 0.049,Y -588.246,Z 1299.172,A 0.000,B 0.000,C 90.000,E1 66.922} C_DIS
LIN {X -0.332,Y -589.333,Z 1299.163,A 0.000,B 0.000,C 90.000,E1 65.357} C_DIS
LIN {X 0.085,Y -590.484,Z 1299.154,A 0.000,B 0.000,C 90.000,E1 63.717} C_DIS
LIN {X 0.054,Y -592.272,Z 1299.142,A 0.000,B 0.000,C 90.000,E1 61.591} C_DIS
LIN {X 0.130,Y -593.563,Z 1299.135,A 0.000,B 0.000,C 90.000,E1 60.255} C_DIS
LIN {X -0.065,Y -594.883,Z 1299.128,A 0.000,B 0.000,C 90.000,E1 58.948} C_DIS
LIN {X -0.101,Y -597.131,Z 1299.116,A 0.000,B 0.000,C 90.000,E1 56.834} C_DIS
LIN {X -0.216,Y -598.762,Z 1299.107,A 0.000,B 0.000,C 90.000,E1 55.261} C_DIS
LIN {X -0.207,Y -600.511,Z 1299.097,A 0.000,B 0.000,C 90.000,E1 53.417} C_DIS
LIN {X 0.208,Y -602.069,Z 1299.086,A 0.000,B 0.000,C 90.000,E1 51.537} C_DIS
LIN {X -0.106,Y -602.867,Z 1299.081,A 0.000,B 0.000,C 90.000,E1 50.517} C_DIS
LIN {X 0.016,Y -603.848,Z 1299.072,A 0.000,B 0.000,C 90.000,E1 48.933} C_DIS
LIN {X 0.106,Y -604.150,Z 1299.066,A 0.000,B 0.000,C 90.000,E1 47.877} C_DIS
LIN {X 0.205,Y -604.484,Z 1299.057,A 0.000,B 0.000,C 90.000,E1 46.296} C_DIS
LIN {X 0.275,Y -604.654,Z 1299.052,A 0.000,B 0.000,C 90.000,E1 45.243} C_DIS
LIN {X 0.346,Y -604.546,Z 1299.046,A 0.000,B 0.000,C 90.000,E1 44.190} C_DIS
LIN {X -0.199,Y -604.187,Z 1299.038,A 0.000,B 0.000,C 90.000,E1 42.933} C_DIS
LIN {X 0.301,Y -603.904,Z 1299.033,A 0.000,B 0.000,C 90.000,E1 41.838} C_DIS
LIN {X 0.144,Y -603.601,Z 1299.028,A 0.000,B 0.000,C 90.000,E1 41.067} C_DIS
LIN {X 0.022,Y -602.999,Z 1299.021,A 0.000,B 0.000,C 90.000,E1 39.769} C_DIS
LIN {X -0.069,Y -602.628,Z 1299.017,A 0.000,B 0.000,C 90.000,E1 38.991} C_DIS
LIN {X 0.221,Y -602.135,Z 1299.012,A 0.000,B 0.000,C 90.000,E1 38.177} C_DIS
LIN {X 0.156,Y -600.902,Z 1299.005,A 0.000,B 0.000,C 90.000,E1 36.870} C_DIS
LIN {X 0.303,Y -599.607,Z 1298.999,A 0.000,B 0.000,C 90.000,E1 35.804} C_DIS
LIN {X 0.191,Y -598.523,Z 1298.995,A 0.000,B 0.000,C 90.000,E1 35.025} C_DIS
LIN {X 0.190,Y -596.279,Z 1298.987,A 0.000,B 0.000,C 90.000,E1 33.706} C_DIS
LIN {X -0.290,Y -594.649,Z 1298.983,A 0.000,B 0.000,C 90.000,E1 32.959} C_DIS
LIN {X -0.177,Y -593.467,Z 1298.980,A 0.000,B 0.000,C 90.000,E1 32.418} C_DIS
LIN {X 0.133,Y -591.343,Z 1298.976,A 0.000,B 0.000,C 90.000,E1 31.592} C_DIS
LIN {X 0.109,Y -588.964,Z 1298.971,A 0.000,B 0.000,C 90.000,E1 30.797} C_DIS
LIN {X -0.004,Y -588.143,Z 1298.970,A 0.000,B 0.000,C 90.000,E1 30.541} C_DIS
LIN {X -0.057,Y -585.168,Z 1298.965,A 0.000,B 0.000,C 90.000,E1 29.745} C_DIS
LIN {X -0.014,Y -583.021,Z 1298.962,A 0.000,B 0.000,C 90.000,E1 29.205} C_DIS
LIN {X -0.127,Y -579.420,Z 1298.958,A 0.000,B 0.000,C 90.000,E1 28.409} C_DIS
LIN {X 0.176,Y -577.478,Z 1298.956,A 0.000,B 0.000,C 90.000,E1 27.975} C_DIS
LIN {X -0.190,Y -573.872,Z 1298.952,A 0.000,B 0.000,C 90.000,E1 27.334} C_DIS
LIN {X 0.101,Y -569.289,Z 1298.947,A 0.000,B 0.000,C 90.000,E1 26.488} C_DIS
LIN {X 0.175,Y -565.000,Z 1298.943,A 0.000,B 0.000,C 90.000,E1 25.796} C_DIS
LIN {X 0.017,Y -558.392,Z 1298.938,A 0.000,B 0.000,C 90.000,E1 24.847} C_DIS
LIN {X 0.000,Y -553.195,Z 1298.934,A 0.000,B 0.000,C 90.000,E1 24.155} C_DIS
LIN {X 0.054,Y -548.711,Z 1298.931,A 0.000,B 0.000,C 90.000,E1 23.590} C_DIS
LIN {X -0.301,Y -545.238,Z 1298.929,A 0.000,B 0.000,C 90.000,E1 23.206} C_DIS
LIN {X -0.209,Y -536.624,Z 1298.923,A 0.000,B 0.000,C 90.000,E1 22.206} C_DIS
LIN {X -0.164,Y -528.812,Z 1298.919,A 0.000,B 0.000,C 90.000,E1 21.354} C_DIS
LIN {X 0.198,Y -520.966,Z 1298.914,A 0.000,B 0.000,C 90.000,E1 20.482} C_DIS
LIN {X -0.070,Y -513.191,Z 1298.909,A 0.000,B 0.000,C 90.000,E1 19.704} C_DIS
LIN {X 0.154,Y -504.964,Z 1298.905,A 0.000,B 0.000,C 90.000,E1 18.852} C_DIS
LIN {X 0.304,Y -495.241,Z 1298.900,A 0.000,B 0.000,C 90.000,E1 17.873} C_DIS
LIN {X -0.144,Y -485.206,Z 1298.894,A 0.000,B 0.000,C 90.000,E1 16.968} C_DIS
LIN {X 0.183,Y -476.508,Z 1298.890,A 0.000,B 0.000,C 90.000,E1 16.134} C_DIS
LIN {X 0.041,Y -463.197,Z 1298.883,A 0.000,B 0.000,C 90.000,E1 14.954} C_DIS
LIN {X 0.117,Y -443.163,Z 1298.873,A 0.000,B 0.000,C 90.000,E1 13.063} C_DIS
LIN {X -0.063,Y -424.389,Z 1298.862,A 0.000,B 0.000,C 90.000,E1 11.186} C_DIS
LIN {X -0.172,Y -408.676,Z 1298.853,A 0.000,B 0.000,C 90.000,E1 9.500} C_DIS
LIN {X 0.032,Y -400.130,Z 1298.847,A 0.000,B 0.000,C 90.000,E1 8.511} C_DIS
LIN {X 0.142,Y -397.406,Z 1298.845,A 0.000,B 0.000,C 90.000,E1 8.163} C_DIS
LIN {X 0.000,Y -395.273,Z 1298.844,A 0.000,B 0.000,C 90.000,E1 7.814} C_DIS
LIN {X -0.038,Y -395.277,Z 1298.843,A 0.000,B 0.000,C 90.000,E1 7.814} C_DIS
LIN {X 0.112,Y -396.105,Z 1298.843,A 0.000,B 0.000,C 90.000,E1 7.644} C_DIS
LIN {X -0.080,Y -399.538,Z 1298.841,A 0.000,B 0.000,C 90.000,E1 7.352} C_DIS
LIN {X -0.103,Y -405.009,Z 1298.839,A 0.000,B 0.000,C 90.000,E1 7.004} C_DIS
LIN {X 0.156,Y -411.407,Z 1298.837,A 0.000,B 0.000,C 90.000,E1 6.606} C_DIS
LIN {X 0.111,Y -419.317,Z 1298.834,A 0.000,B 0.000,C 90.000,E1 6.087} C_DIS
LIN {X 0.137,Y -428.722,Z 1298.830,A 0.000,B 0.000,C 90.000,E1 5.391} C_DIS
LIN {X -0.136,Y -436.358,Z 1298.827,A 0.000,B 0.000,C 90.000,E1 4.821} C_DIS
LIN {X 0.123,Y -445.478,Z 1298.822,A 0.000,B 0.000,C 90.000,E1 4.012} C_DIS
LIN {X 0.083,Y -454.383,Z 1298.818,A 0.000,B 0.000,C 90.000,E1 3.212} C_DIS
LIN {X 0.042,Y -461.540,Z 1298.814,A 0.000,B 0.000,C 90.000,E1 2.522} C_DIS
LIN {X 0.034,Y -467.029,Z 1298.811,A 0.000,B 0.000,C 90.000,E1 1.949} C_DIS
LIN {X 0.236,Y -473.508,Z 1298.807,A 0.000,B 0.000,C 90.000,E1 1.203} C_DIS
LIN {X -0.026,Y -479.688,Z 1298.803,A 0.000,B 0.000,C 90.000,E1 0.458} C_DIS
LIN {X 0.000,Y -483.113,Z 1298.800,A 0.000,B 0.000,C 90.000,E1 360.000} C_DIS
LIN {X 0.159,Y -487.928,Z 1298.796,A 0.000,B 0.000,C 90.000,E1 359.312} C_DIS
LIN {X -0.009,Y -492.931,Z 1298.792,A 0.000,B 0.000,C 90.000,E1 358.568} C_DIS
LIN {X 0.204,Y -496.790,Z 1298.789,A 0.000,B 0.000,C 90.000,E1 357.936} C_DIS
LIN {X -0.199,Y -501.949,Z 1298.784,A 0.000,B 0.000,C 90.000,E1 357.078} C_DIS
LIN {X 0.090,Y -505.235,Z 1298.780,A 0.000,B 0.000,C 90.000,E1 356.445} C_DIS
LIN {X -0.200,Y -509.819,Z 1298.775,A 0.000,B 0.000,C 90.000,E1 355.584} C_DIS
LIN {X 0.156,Y -512.684,Z 1298.772,A 0.000,B 0.000,C 90.000,E1 354.951} C_DIS
LIN {X 0.026,Y -515.414,Z 1298.769,A 0.000,B 0.000,C 90.000,E1 354.375} C_DIS
LIN {X -0.086,Y -517.983,Z 1298.766,A 0.000,B 0.000,C 90.000,E1 353.799} C_DIS
LIN {X -0.182,Y -520.399,Z 1298.762,A 0.000,B 0.000,C 90.000,E1 353.223} C_DIS
LIN {X 0.252,Y -523.739,Z 1298.757,A 0.000,B 0.000,C 90.000,E1 352.299} C_DIS
LIN {X 0.192,Y -525.859,Z 1298.754,A 0.000,B 0.000,C 90.000,E1 351.724} C_DIS
LIN {X 0.186,Y -529.606,Z 1298.748,A 0.000,B 0.000,C 90.000,E1 350.566} C_DIS
LIN {X -0.239,Y -532.151,Z 1298.743,A 0.000,B 0.000,C 90.000,E1 349.746} C_DIS
LIN {X -0.058,Y -535.197,Z 1298.737,A 0.000,B 0.000,C 90.000,E1 348.578} C_DIS
LIN {X 0.107,Y -537.198,Z 1298.732,A 0.000,B 0.000,C 90.000,E1 347.701} C_DIS
LIN {X -0.232,Y -538.919,Z 1298.727,A 0.000,B 0.000,C 90.000,E1 346.881} C_DIS
LIN {X 0.166,Y -540.904,Z 1298.721,A 0.000,B 0.000,C 90.000,E1 345.700} C_DIS
LIN {X -0.004,Y -542.153,Z 1298.716,A 0.000,B 0.000,C 90.000,E1 344.866} C_DIS
LIN {X -0.158,Y -543.126,Z 1298.711,A 0.000,B 0.000,C 90.000,E1 344.031} C_DIS
LIN {X -0.228,Y -544.108,Z 1298.705,A 0.000,B 0.000,C 90.000,E1 342.906} C_DIS
LIN {X -0.203,Y -544.578,Z 1298.700,A 0.000,B 0.000,C 90.000,E1 342.054} C_DIS
LIN {X 0.175,Y -544.714,Z 1298.696,A 0.000,B 0.000,C 90.000,E1 341.167} C_DIS
LIN {X -0.305,Y -544.540,Z 1298.691,A 0.000,B 0.000,C 90.000,E1 340.369} C_DIS
LIN {X -0.271,Y -544.075,Z 1298.686,A 0.000,B 0.000,C 90.000,E1 339.518} C_DIS
LIN {X -0.048,Y -543.368,Z 1298.681,A 0.000,B 0.000,C 90.000,E1 338.646} C_DIS
LIN {X -0.269,Y -542.601,Z 1298.678,A 0.000,B 0.000,C 90.000,E1 338.103} C_DIS
LIN {X 0.176,Y -540.961,Z 1298.672,A 0.000,B 0.000,C 90.000,E1 336.922} C_DIS
LIN {X -0.089,Y -540.458,Z 1298.670,A 0.000,B 0.000,C 90.000,E1 336.666} C_DIS
LIN {X 0.100,Y -538.454,Z 1298.666,A 0.000,B 0.000,C 90.000,E1 335.793} C_DIS
LIN {X -0.293,Y -534.598,Z 1298.658,A 0.000,B 0.000,C 90.000,E1 334.409} C_DIS
LIN {X 0.054,Y -531.788,Z 1298.653,A 0.000,B 0.000,C 90.000,E1 333.512} C_DIS
LIN {X 0.071,Y -528.094,Z 1298.646,A 0.000,B 0.000,C 90.000,E1 332.359} C_DIS
LIN {X -0.125,Y -525.067,Z 1298.642,A 0.000,B 0.000,C 90.000,E1 331.513} C_DIS
LIN {X 0.200,Y -521.035,Z 1298.636,A 0.000,B 0.000,C 90.000,E1 330.461} C_DIS
LIN {X 0.088,Y -517.890,Z 1298.632,A 0.000,B 0.000,C 90.000,E1 329.744} C_DIS
LIN {X -0.050,Y -512.278,Z 1298.625,A 0.000,B 0.000,C 90.000,E1 328.584} C_DIS
LIN {X -0.245,Y -508.636,Z 1298.621,A 0.000,B 0.000,C 90.000,E1 327.867} C_DIS
LIN {X -0.123,Y -504.412,Z 1298.616,A 0.000,B 0.000,C 90.000,E1 326.962} C_DIS
LIN {X -0.120,Y -501.346,Z 1298.612,A 0.000,B 0.000,C 90.000,E1 326.215} C_DIS
LIN {X 0.056,Y -499.301,Z 1298.609,A 0.000,B 0.000,C 90.000,E1 325.595} C_DIS
LIN {X 0.198,Y -497.127,Z 1298.604,A 0.000,B 0.000,C 90.000,E1 324.689} C_DIS
LIN {X 0.200,Y -495.626,Z 1298.599,A 0.000,B 0.000,C 90.000,E1 323.783} C_DIS
LIN {X 0.195,Y -494.239,Z 1298.591,A 0.000,B 0.000,C 90.000,E1 322.271} C_DIS
LIN {X -0.075,Y -493.772,Z 1298.584,A 0.000,B 0.000,C 90.000,E1 321.090} C_DIS
LIN {X 0.239,Y -493.862,Z 1298.569,A 0.000,B 0.000,C 90.000,E1 318.324} C_DIS
LIN {X 0.097,Y -494.022,Z 1298.560,A 0.000,B 0.000,C 90.000,E1 316.824} C_DIS
LIN {X 0.297,Y -493.876,Z 1298.555,A 0.000,B 0.000,C 90.000,E1 315.891} C_DIS
LIN {X -0.041,Y -493.541,Z 1298.552,A 0.000,B 0.000,C 90.000,E1 315.324} C_DIS
LIN {X -0.033,Y -492.920,Z 1298.548,A 0.000,B 0.000,C 90.000,E1 314.717} C_DIS
LIN {X -0.025,Y -491.938,Z 1298.545,A 0.000,B 0.000,C 90.000,E1 314.109} C_DIS
LIN {X 0.147,Y -491.218,Z 1298.543,A 0.000,B 0.000,C 90.000,E1 313.785} C_DIS
LIN {X -0.020,Y -490.198,Z 1298.542,A 0.000,B 0.000,C 90.000,E1 313.500} C_DIS
LIN {X 0.065,Y -489.451,Z 1298.541,A 0.000,B 0.000,C 90.000,E1 313.338} C_DIS
LIN {X -0.304,Y -484.652,Z 1298.537,A 0.000,B 0.000,C 90.000,E1 312.771} C_DIS
LIN {X -0.018,Y -466.114,Z 1298.524,A 0.000,B 0.000,C 90.000,E1 310.253} C_DIS
LIN {X -0.231,Y -449.339,Z 1298.510,A 0.000,B 0.000,C 90.000,E1 307.729} C_DIS
LIN {X -0.148,Y -434.215,Z 1298.495,A 0.000,B 0.000,C 90.000,E1 305.105} C_DIS
LIN {X -0.059,Y -420.642,Z 1298.480,A 0.000,B 0.000,C 90.000,E1 302.418} C_DIS
LIN {X -0.226,Y -407.820,Z 1298.464,A 0.000,B 0.000,C 90.000,E1 299.539} C_DIS
LIN {X -0.037,Y -397.876,Z 1298.450,A 0.000,B 0.000,C 90.000,E1 296.924} C_DIS
LIN {X -0.076,Y -397.873,Z 1298.450,A 0.000,B 0.000,C 90.000,E1 296.924} C_DIS
LIN {X 0.110,Y -401.434,Z 1298.427,A 0.000,B 0.000,C 90.000,E1 292.845} C_DIS
LIN {X -0.024,Y -401.673,Z 1298.425,A 0.000,B 0.000,C 90.000,E1 292.514} C_DIS
LIN {X 0.107,Y -404.763,Z 1298.394,A 0.000,B 0.000,C 90.000,E1 286.913} C_DIS
LIN {X 0.013,Y -406.154,Z 1298.363,A 0.000,B 0.000,C 90.000,E1 281.366} C_DIS
LIN {X 0.118,Y -405.645,Z 1298.334,A 0.000,B 0.000,C 90.000,E1 276.144} C_DIS
LIN {X 0.122,Y -405.635,Z 1298.332,A 0.000,B 0.000,C 90.000,E1 275.796} C_DIS
LIN {X 0.195,Y -403.556,Z 1298.305,A 0.000,B 0.000,C 90.000,E1 270.917} C_DIS
LIN {X 0.130,Y -403.092,Z 1298.301,A 0.000,B 0.000,C 90.000,E1 270.229} C_DIS
LIN {X -0.043,Y -399.030,Z 1298.272,A 0.000,B 0.000,C 90.000,E1 265.008} C_DIS
LIN {X -0.126,Y -398.169,Z 1298.268,A 0.000,B 0.000,C 90.000,E1 264.318} C_DIS
LIN {X 0.127,Y -392.958,Z 1298.241,A 0.000,B 0.000,C 90.000,E1 259.342} C_DIS
LIN {X 0.085,Y -392.533,Z 1298.239,A 0.000,B 0.000,C 90.000,E1 258.993} C_DIS
LIN {X -0.140,Y -386.158,Z 1298.213,A 0.000,B 0.000,C 90.000,E1 254.393} C_DIS
LIN {X -0.177,Y -385.044,Z 1298.207,A 0.000,B 0.000,C 90.000,E1 253.323} C_DIS
LIN {X 0.069,Y -379.007,Z 1298.187,A 0.000,B 0.000,C 90.000,E1 249.571} C_DIS
LIN {X 0.032,Y -379.020,Z 1298.187,A 0.000,B 0.000,C 90.000,E1 249.571} C_DIS
LIN {X 0.036,Y -387.776,Z 1298.169,A 0.000,B 0.000,C 90.000,E1 246.433} C_DIS
LIN {X -0.115,Y -398.403,Z 1298.151,A 0.000,B 0.000,C 90.000,E1 243.256} C_DIS
LIN {X 0.134,Y -409.968,Z 1298.135,A 0.000,B 0.000,C 90.000,E1 240.255} C_DIS
LIN {X -0.061,Y -423.114,Z 1298.119,A 0.000,B 0.000,C 90.000,E1 237.375} C_DIS
LIN {X -0.002,Y -437.020,Z 1298.104,A 0.000,B 0.000,C 90.000,E1 234.689} C_DIS
LIN {X -0.017,Y -450.485,Z 1298.091,A 0.000,B 0.000,C 90.000,E1 232.396} C_DIS
LIN {X -0.302,Y -451.369,Z 1298.090,A 0.000,B 0.000,C 90.000,E1 232.271} C_DIS
LIN {X 0.045,Y -451.972,Z 1298.089,A 0.000,B 0.000,C 90.000,E1 232.065} C_DIS
LIN {X 0.035,Y -452.800,Z 1298.088,A 0.000,B 0.000,C 90.000,E1 231.743} C_DIS
LIN {X 0.104,Y -453.369,Z 1298.086,A 0.000,B 0.000,C 90.000,E1 231.412} C_DIS
LIN {X -0.179,Y -454.092,Z 1298.082,A 0.000,B 0.000,C 90.000,E1 230.803} C_DIS
LIN {X -0.103,Y -454.472,Z 1298.079,A 0.000,B 0.000,C 90.000,E1 230.150} C_DIS
LIN {X 0.267,Y -454.623,Z 1298.075,A 0.000,B 0.000,C 90.000,E1 229.461} C_DIS
LIN {X 0.018,Y -454.540,Z 1298.070,A 0.000,B 0.000,C 90.000,E1 228.528} C_DIS
LIN {X -0.108,Y -453.940,Z 1298.055,A 0.000,B 0.000,C 90.000,E1 225.972} C_DIS
LIN {X 0.026,Y -453.766,Z 1298.043,A 0.000,B 0.000,C 90.000,E1 223.704} C_DIS
LIN {X -0.133,Y -455.426,Z 1298.012,A 0.000,B 0.000,C 90.000,E1 218.257} C_DIS
LIN {X 0.148,Y -456.753,Z 1298.002,A 0.000,B 0.000,C 90.000,E1 216.297} C_DIS
LIN {X -0.123,Y -459.181,Z 1297.986,A 0.000,B 0.000,C 90.000,E1 213.452} C_DIS
LIN {X -0.048,Y -462.605,Z 1297.968,A 0.000,B 0.000,C 90.000,E1 210.256} C_DIS
LIN {X -0.232,Y -464.653,Z 1297.959,A 0.000,B 0.000,C 90.000,E1 208.693} C_DIS
LIN {X 0.118,Y -467.560,Z 1297.947,A 0.000,B 0.000,C 90.000,E1 206.437} C_DIS
LIN {X -0.037,Y -470.310,Z 1297.937,A 0.000,B 0.000,C 90.000,E1 204.567} C_DIS
LIN {X -0.072,Y -472.574,Z 1297.928,A 0.000,B 0.000,C 90.000,E1 203.003} C_DIS
LIN {X 0.116,Y -476.267,Z 1297.914,A 0.000,B 0.000,C 90.000,E1 200.482} C_DIS
LIN {X 0.283,Y -479.177,Z 1297.904,A 0.000,B 0.000,C 90.000,E1 198.598} C_DIS
LIN {X -0.086,Y -481.642,Z 1297.895,A 0.000,B 0.000,C 90.000,E1 197.094} C_DIS
LIN {X -0.082,Y -484.145,Z 1297.886,A 0.000,B 0.000,C 90.000,E1 195.552} C_DIS
LIN {X -0.025,Y -486.585,Z 1297.878,A 0.000,B 0.000,C 90.000,E1 194.008} C_DIS
LIN {X 0.076,Y -488.589,Z 1297.871,A 0.000,B 0.000,C 90.000,E1 192.771} C_DIS
LIN {X -0.014,Y -491.483,Z 1297.861,A 0.000,B 0.000,C 90.000,E1 190.950} C_DIS
LIN {X -0.227,Y -494.373,Z 1297.851,A 0.000,B 0.000,C 90.000,E1 189.151} C_DIS
LIN {X 0.116,Y -497.216,Z 1297.841,A 0.000,B 0.000,C 90.000,E1 187.296} C_DIS
LIN {X -0.096,Y -500.023,Z 1297.831,A 0.000,B 0.000,C 90.000,E1 185.511} C_DIS
LIN {X 0.093,Y -501.351,Z 1297.826,A 0.000,B 0.000,C 90.000,E1 184.588} C_DIS
LIN {X -0.073,Y -503.893,Z 1297.816,A 0.000,B 0.000,C 90.000,E1 182.808} C_DIS
LIN {X 0.004,Y -505.410,Z 1297.809,A 0.000,B 0.000,C 90.000,E1 181.604} C_DIS
LIN {X -0.008,Y -507.139,Z 1297.801,A 0.000,B 0.000,C 90.000,E1 180.115} C_DIS
LIN {X 0.204,Y -508.131,Z 1297.796,A 0.000,B 0.000,C 90.000,E1 179.198} C_DIS
LIN {X -0.161,Y -509.128,Z 1297.789,A 0.000,B 0.000,C 90.000,E1 178.051} C_DIS
LIN {X 0.002,Y -510.058,Z 1297.782,A 0.000,B 0.000,C 90.000,E1 176.846} C_DIS
LIN {X 0.176,Y -510.797,Z 1297.776,A 0.000,B 0.000,C 90.000,E1 175.641} C_DIS
LIN {X 0.031,Y -511.054,Z 1297.773,A 0.000,B 0.000,C 90.000,E1 175.065} C_DIS
LIN {X 0.256,Y -511.304,Z 1297.766,A 0.000,B 0.000,C 90.000,E1 173.856} C_DIS
LIN {X -0.027,Y -511.351,Z 1297.760,A 0.000,B 0.000,C 90.000,E1 172.704} C_DIS
LIN {X -0.210,Y -511.145,Z 1297.755,A 0.000,B 0.000,C 90.000,E1 171.837} C_DIS
LIN {X 0.188,Y -510.667,Z 1297.750,A 0.000,B 0.000,C 90.000,E1 170.905} C_DIS
LIN {X -0.042,Y -509.797,Z 1297.743,A 0.000,B 0.000,C 90.000,E1 169.746} C_DIS
LIN {X -0.157,Y -508.891,Z 1297.738,A 0.000,B 0.000,C 90.000,E1 168.870} C_DIS
LIN {X 0.217,Y -507.626,Z 1297.733,A 0.000,B 0.000,C 90.000,E1 167.937} C_DIS
LIN {X 0.138,Y -505.662,Z 1297.727,A 0.000,B 0.000,C 90.000,E1 166.756} C_DIS
LIN {X 0.036,Y -503.270,Z 1297.720,A 0.000,B 0.000,C 90.000,E1 165.574} C_DIS
LIN {X -0.207,Y -498.516,Z 1297.708,A 0.000,B 0.000,C 90.000,E1 163.504} C_DIS
LIN {X -0.188,Y -496.366,Z 1297.703,A 0.000,B 0.000,C 90.000,E1 162.598} C_DIS
LIN {X 0.165,Y -492.860,Z 1297.697,A 0.000,B 0.000,C 90.000,E1 161.348} C_DIS
LIN {X 0.146,Y -489.319,Z 1297.690,A 0.000,B 0.000,C 90.000,E1 160.134} C_DIS
LIN {X 0.224,Y -486.166,Z 1297.685,A 0.000,B 0.000,C 90.000,E1 159.209} C_DIS
LIN {X -0.178,Y -483.561,Z 1297.680,A 0.000,B 0.000,C 90.000,E1 158.337} C_DIS
LIN {X -0.167,Y -482.982,Z 1297.678,A 0.000,B 0.000,C 90.000,E1 158.028} C_DIS
LIN {X -0.160,Y -482.665,Z 1297.676,A 0.000,B 0.000,C 90.000,E1 157.720} C_DIS
LIN {X -0.152,Y -482.846,Z 1297.673,A 0.000,B 0.000,C 90.000,E1 157.102} C_DIS
LIN {X -0.146,Y -484.194,Z 1297.669,A 0.000,B 0.000,C 90.000,E1 156.485} C_DIS
LIN {X -0.142,Y -485.744,Z 1297.668,A 0.000,B 0.000,C 90.000,E1 156.177} C_DIS
LIN {X 0.085,Y -486.457,Z 1297.667,A 0.000,B 0.000,C 90.000,E1 155.997} C_DIS
LIN {X -0.134,Y -487.796,Z 1297.666,A 0.000,B 0.000,C 90.000,E1 155.869} C_DIS
LIN {X 0.117,Y -490.104,Z 1297.664,A 0.000,B 0.000,C 90.000,E1 155.537} C_DIS
LIN {X -0.120,Y -493.235,Z 1297.663,A 0.000,B 0.000,C 90.000,E1 155.281} C_DIS
LIN {X -0.143,Y -494.412,Z 1297.662,A 0.000,B 0.000,C 90.000,E1 155.153} C_DIS
LIN {X -0.036,Y -500.620,Z 1297.659,A 0.000,B 0.000,C 90.000,E1 154.537} C_DIS
LIN {X -0.275,Y -504.780,Z 1297.656,A 0.000,B 0.000,C 90.000,E1 154.152} C_DIS
LIN {X 0.257,Y -511.207,Z 1297.652,A 0.000,B 0.000,C 90.000,E1 153.384} C_DIS
LIN {X -0.249,Y -514.968,Z 1297.650,A 0.000,B 0.000,C 90.000,E1 152.999} C_DIS
LIN {X -0.129,Y -519.488,Z 1297.647,A 0.000,B 0.000,C 90.000,E1 152.410} C_DIS
LIN {X -0.056,Y -523.656,Z 1297.643,A 0.000,B 0.000,C 90.000,E1 151.820} C_DIS
LIN {X -0.231,Y -527.365,Z 1297.640,A 0.000,B 0.000,C 90.000,E1 151.257} C_DIS
LIN {X -0.130,Y -530.497,Z 1297.637,A 0.000,B 0.000,C 90.000,E1 150.667} C_DIS
LIN {X -0.005,Y -533.092,Z 1297.634,A 0.000,B 0.000,C 90.000,E1 150.078} C_DIS
LIN {X 0.264,Y -535.941,Z 1297.630,A 0.000,B 0.000,C 90.000,E1 149.331} C_DIS
LIN {X 0.118,Y -536.717,Z 1297.629,A 0.000,B 0.000,C 90.000,E1 149.203} C_DIS
LIN {X -0.032,Y -538.353,Z 1297.627,A 0.000,B 0.000,C 90.000,E1 148.791} C_DIS
LIN {X -0.174,Y -539.341,Z 1297.626,A 0.000,B 0.000,C 90.000,E1 148.663} C_DIS
LIN {X -0.314,Y -540.112,Z 1297.625,A 0.000,B 0.000,C 90.000,E1 148.535} C_DIS
LIN {X 0.078,Y -540.800,Z 1297.624,A 0.000,B 0.000,C 90.000,E1 148.280} C_DIS
LIN {X 0.151,Y -541.344,Z 1297.624,A 0.000,B 0.000,C 90.000,E1 148.201} C_DIS
LIN {X 0.013,Y -542.634,Z 1297.623,A 0.000,B 0.000,C 90.000,E1 148.074} C_DIS
LIN {X 0.050,Y -544.577,Z 1297.621,A 0.000,B 0.000,C 90.000,E1 147.788} C_DIS
LIN {X -0.075,Y -550.077,Z 1297.619,A 0.000,B 0.000,C 90.000,E1 147.454} C_DIS
LIN {X -0.089,Y -556.452,Z 1297.617,A 0.000,B 0.000,C 90.000,E1 147.089} C_DIS
LIN {X -0.101,Y -562.317,Z 1297.615,A 0.000,B 0.000,C 90.000,E1 146.707} C_DIS
LIN {X -0.109,Y -571.463,Z 1297.612,A 0.000,B 0.000,C 90.000,E1 146.087} C_DIS
LIN {X -0.300,Y -577.159,Z 1297.609,A 0.000,B 0.000,C 90.000,E1 145.674} C_DIS
LIN {X -0.221,Y -586.965,Z 1297.605,A 0.000,B 0.000,C 90.000,E1 144.895} C_DIS
LIN {X -0.023,Y -592.215,Z 1297.602,A 0.000,B 0.000,C 90.000,E1 144.402} C_DIS
LIN {X -0.031,Y -597.168,Z 1297.599,A 0.000,B 0.000,C 90.000,E1 143.909} C_DIS
LIN {X 0.088,Y -600.709,Z 1297.598,A 0.000,B 0.000,C 90.000,E1 143.543} C_DIS
